C05460=1089.469,232.311,-75.849,176.386,20.960,153.192
C05461=1089.476,232.559,-75.874,176.389,20.962,153.192
C05462=1089.481,232.808,-75.901,176.392,20.965,153.192
C05463=1089.486,233.056,-75.926,176.394,20.967,153.192
C05464=1089.492,233.305,-75.952,176.398,20.970,153.192
C05465=1089.498,233.554,-75.977,176.400,20.972,153.192
C05466=1089.504,233.802,-76.004,176.403,20.974,153.192
C05467=1089.509,234.051,-76.030,176.406,20.977,153.192
C05468=1089.514,234.299,-76.056,176.409,20.979,153.192
C05469=1089.520,234.547,-76.082,176.412,20.981,153.192
C05470=1089.525,234.796,-76.108,176.414,20.984,153.192
C05471=1089.531,235.045,-76.134,176.417,20.986,153.192
C05472=1089.537,235.294,-76.160,176.420,20.989,153.192
C05473=1089.545,235.671,-76.200,176.424,20.992,153.193
C05474=1089.554,236.049,-76.239,176.429,20.996,153.193
C05475=1089.562,236.426,-76.279,176.433,20.999,153.193
C05476=1089.571,236.805,-76.319,176.437,21.003,153.193
C05477=1089.577,237.053,-76.345,176.440,21.006,153.193
C05478=1089.583,237.302,-76.371,176.443,21.008,153.193
C05479=1089.588,237.551,-76.397,176.445,21.010,153.193
C05480=1089.593,237.798,-76.424,176.448,21.013,153.193
C05481=1089.599,238.047,-76.449,176.452,21.015,153.193
C05482=1089.605,238.296,-76.476,176.454,21.017,153.193
C05483=1089.610,238.545,-76.502,176.457,21.020,153.193
C05484=1089.616,238.793,-76.529,176.459,21.022,153.193
C05485=1089.621,239.042,-76.555,176.463,21.025,153.193
C05486=1089.627,239.290,-76.581,176.466,21.027,153.193
C05487=1089.633,239.539,-76.607,176.468,21.029,153.194
C05488=1089.638,239.788,-76.634,176.471,21.032,153.194
C05489=1089.644,240.036,-76.661,176.475,21.034,153.194
C05490=1089.650,240.285,-76.686,176.477,21.036,153.194
C05491=1089.655,240.533,-76.713,176.480,21.039,153.194
C05492=1089.661,240.782,-76.739,176.483,21.042,153.194
C05493=1089.667,241.031,-76.766,176.486,21.043,153.194
C05494=1089.672,241.279,-76.792,176.489,21.046,153.194
C05495=1089.678,241.527,-76.819,176.491,21.048,153.194
C05496=1089.684,241.776,-76.845,176.494,21.051,153.194
C05497=1089.689,242.025,-76.872,176.497,21.054,153.194
C05498=1089.695,242.273,-76.898,176.500,21.056,153.194
C05499=1089.701,242.522,-76.924,176.503,21.058,153.194
C05500=1089.706,242.770,-76.951,176.506,21.060,153.194
C05501=1089.712,243.019,-76.977,176.508,21.063,153.195
C05502=1089.718,243.267,-77.004,176.511,21.065,153.195
C05503=1089.724,243.516,-77.031,176.515,21.068,153.195
C05504=1089.729,243.765,-77.057,176.517,21.070,153.195
C05505=1089.734,244.013,-77.084,176.520,21.073,153.195
C05506=1089.740,244.262,-77.111,176.523,21.075,153.195
C05507=1089.746,244.510,-77.137,176.526,21.077,153.195
C05508=1089.752,244.758,-77.164,176.529,21.080,153.195
C05509=1089.757,245.007,-77.191,176.532,21.083,153.195
C05510=1089.762,245.256,-77.217,176.534,21.085,153.195
C05511=1089.768,245.504,-77.244,176.537,21.088,153.195
C05512=1089.774,245.753,-77.270,176.540,21.090,153.195
C05513=1089.779,246.001,-77.297,176.543,21.092,153.195
C05514=1089.784,246.250,-77.324,176.546,21.095,153.196
C05515=1089.790,246.498,-77.351,176.549,21.097,153.196
C05516=1089.796,246.746,-77.377,176.551,21.099,153.196
C05517=1089.802,246.996,-77.405,176.554,21.102,153.196
C05518=1089.807,247.244,-77.432,176.558,21.104,153.196
C05519=1089.813,247.492,-77.458,176.560,21.107,153.196
C05520=1089.818,247.741,-77.486,176.563,21.109,153.196
C05521=1089.824,247.989,-77.512,176.566,21.112,153.196
C05522=1089.830,248.238,-77.539,176.569,21.115,153.196
C05523=1089.835,248.487,-77.566,176.572,21.117,153.196
C05524=1089.841,248.735,-77.593,176.575,21.119,153.196
C05525=1089.849,249.106,-77.634,176.579,21.123,153.196
C05526=1089.857,249.476,-77.674,176.583,21.127,153.197
C05527=1089.865,249.847,-77.714,176.588,21.131,153.197
C05528=1089.874,250.218,-77.754,176.592,21.134,153.197
C05529=1089.879,250.467,-77.782,176.595,21.137,153.197
C05530=1089.885,250.715,-77.808,176.597,21.139,153.197
C05531=1089.890,250.963,-77.836,176.601,21.142,153.197
C05532=1089.896,251.212,-77.863,176.604,21.145,153.197
C05533=1089.901,251.460,-77.890,176.607,21.147,153.197
C05534=1089.907,251.710,-77.917,176.609,21.149,153.197
C05535=1089.912,251.958,-77.944,176.612,21.152,153.197
C05536=1089.918,252.206,-77.972,176.615,21.155,153.198
C05537=1089.923,252.455,-77.999,176.618,21.157,153.198
C05538=1089.929,252.703,-78.026,176.621,21.160,153.198
C05539=1089.934,252.951,-78.054,176.624,21.162,153.198
C05540=1089.941,253.200,-78.081,176.627,21.164,153.198
C05541=1089.946,253.449,-78.108,176.629,21.167,153.198
C05542=1089.952,253.696,-78.135,176.633,21.169,153.198
C05543=1089.957,253.945,-78.163,176.636,21.172,153.198
C05544=1089.963,254.194,-78.190,176.639,21.175,153.198
C05545=1089.969,254.442,-78.218,176.641,21.177,153.198
C05546=1089.974,254.691,-78.244,176.644,21.179,153.198
C05547=1089.980,254.939,-78.272,176.647,21.182,153.199
C05548=1089.986,255.187,-78.299,176.650,21.184,153.199
C05549=1089.991,255.436,-78.326,176.653,21.187,153.199
C05550=1089.996,255.684,-78.354,176.656,21.190,153.199
C05551=1090.002,255.933,-78.381,176.659,21.192,153.199
C05552=1090.008,256.182,-78.409,176.661,21.194,153.199
C05553=1090.014,256.430,-78.436,176.665,21.197,153.199
C05554=1090.019,256.678,-78.464,176.668,21.200,153.199
C05555=1090.024,256.927,-78.491,176.671,21.202,153.199
C05556=1090.031,257.175,-78.519,176.673,21.205,153.199
C05557=1090.036,257.424,-78.546,176.676,21.207,153.199
C05558=1090.042,257.671,-78.573,176.679,21.210,153.200
C05559=1090.048,257.921,-78.601,176.683,21.212,153.200
C05560=1090.053,258.169,-78.629,176.685,21.215,153.200
C05561=1090.059,258.417,-78.656,176.688,21.217,153.200
C05562=1090.065,258.666,-78.684,176.691,21.219,153.200
C05563=1090.070,258.914,-78.712,176.694,21.222,153.200
C05564=1090.076,259.162,-78.739,176.697,21.224,153.200
C05565=1090.082,259.411,-78.767,176.700,21.227,153.200
C05566=1090.088,259.659,-78.794,176.703,21.230,153.200
C05567=1090.094,259.908,-78.823,176.706,21.232,153.200
C05568=1090.099,260.156,-78.850,176.709,21.235,153.200
C05569=1090.105,260.404,-78.877,176.711,21.237,153.201
C05570=1090.111,260.653,-78.906,176.715,21.240,153.201
C05571=1090.116,260.902,-78.933,176.718,21.242,153.201
C05572=1090.123,261.150,-78.961,176.721,21.245,153.201
C05573=1090.128,261.398,-78.989,176.723,21.247,153.201
C05574=1090.133,261.646,-79.016,176.726,21.250,153.201
C05575=1090.139,261.895,-79.045,176.730,21.252,153.201
C05576=1090.145,262.143,-79.071,176.733,21.255,153.201
C05577=1090.153,262.511,-79.114,176.736,21.259,153.201
C05578=1090.163,262.879,-79.155,176.741,21.262,153.201
C05579=1090.171,263.247,-79.195,176.746,21.266,153.202
C05580=1090.179,263.615,-79.237,176.750,21.270,153.202
C05581=1090.185,263.863,-79.265,176.753,21.273,153.202
C05582=1090.191,264.112,-79.293,176.756,21.275,153.202
C05583=1090.197,264.360,-79.320,176.759,21.277,153.202
C05584=1090.203,264.609,-79.349,176.762,21.280,153.202
C05585=1090.208,264.857,-79.377,176.765,21.283,153.202
C05586=1090.214,265.106,-79.405,176.768,21.285,153.202
C05587=1090.219,265.354,-79.433,176.771,21.288,153.202
C05588=1090.225,265.602,-79.461,176.773,21.290,153.203
C05589=1090.230,265.850,-79.489,176.776,21.293,153.203
C05590=1090.236,266.098,-79.517,176.779,21.296,153.203
C05591=1090.242,266.347,-79.546,176.783,21.298,153.203
C05592=1090.247,266.595,-79.574,176.786,21.301,153.203
C05593=1090.253,266.844,-79.602,176.789,21.304,153.203
C05594=1090.258,267.092,-79.630,176.791,21.306,153.203
C05595=1090.264,267.341,-79.658,176.794,21.309,153.203
C05596=1090.270,267.589,-79.686,176.797,21.311,153.203
C05597=1090.276,267.837,-79.715,176.800,21.314,153.204
C05598=1090.281,268.085,-79.743,176.803,21.317,153.204
C05599=1090.287,268.334,-79.771,176.806,21.319,153.204
C05600=1090.293,268.582,-79.799,176.809,21.322,153.204
C05601=1090.299,268.831,-79.828,176.812,21.325,153.204
C05602=1090.304,269.079,-79.856,176.815,21.327,153.204
C05603=1090.310,269.327,-79.885,176.818,21.330,153.204
C05604=1090.316,269.576,-79.913,176.822,21.332,153.204
C05605=1090.321,269.824,-79.941,176.824,21.335,153.204
C05606=1090.327,270.073,-79.970,176.827,21.337,153.205
C05607=1090.332,270.320,-79.999,176.830,21.340,153.205
C05608=1090.338,270.569,-80.027,176.833,21.343,153.205
C05609=1090.344,270.817,-80.055,176.836,21.346,153.205
C05610=1090.349,271.066,-80.083,176.839,21.348,153.205
C05611=1090.355,271.313,-80.112,176.841,21.350,153.205
C05612=1090.360,271.562,-80.141,176.845,21.353,153.205
C05613=1090.366,271.811,-80.169,176.848,21.356,153.205
C05614=1090.372,272.058,-80.198,176.851,21.359,153.206
C05615=1090.378,272.307,-80.226,176.854,21.362,153.206
C05616=1090.383,272.554,-80.255,176.857,21.364,153.206
C05617=1090.389,272.803,-80.283,176.860,21.367,153.206
C05618=1090.395,273.052,-80.312,176.862,21.369,153.206
C05619=1090.400,273.300,-80.341,176.865,21.372,153.206
C05620=1090.406,273.548,-80.369,176.869,21.375,153.206
C05621=1090.412,273.796,-80.398,176.872,21.377,153.206
C05622=1090.417,274.045,-80.427,176.875,21.380,153.207
C05623=1090.423,274.293,-80.456,176.878,21.383,153.207
C05624=1090.429,274.541,-80.484,176.881,21.386,153.207
C05625=1090.434,274.790,-80.513,176.883,21.388,153.207
C05626=1090.440,275.038,-80.542,176.886,21.391,153.207
C05627=1090.446,275.286,-80.570,176.889,21.394,153.207
C05628=1090.451,275.535,-80.599,176.893,21.396,153.207
C05629=1090.460,275.905,-80.642,176.897,21.400,153.208
C05630=1090.468,276.275,-80.685,176.902,21.405,153.208
C05631=1090.477,276.646,-80.729,176.906,21.408,153.208
C05632=1090.485,277.018,-80.771,176.910,21.412,153.208
C05633=1090.491,277.266,-80.801,176.913,21.415,153.208
C05634=1090.496,277.514,-80.829,176.916,21.418,153.209
C05635=1090.502,277.763,-80.858,176.920,21.421,153.209
C05636=1090.508,278.011,-80.887,176.923,21.423,153.209
C05637=1090.514,278.258,-80.916,176.926,21.426,153.209
C05638=1090.519,278.507,-80.946,176.928,21.429,153.209
C05639=1090.525,278.755,-80.974,176.931,21.432,153.209
C05640=1090.530,279.003,-81.003,176.934,21.435,153.209
C05641=1090.536,279.251,-81.032,176.937,21.437,153.209
C05642=1090.542,279.500,-81.062,176.940,21.440,153.210
C05643=1090.548,279.748,-81.090,176.943,21.443,153.210
C05644=1090.553,279.996,-81.119,176.946,21.446,153.210
C05645=1090.559,280.244,-81.149,176.949,21.448,153.210
C05646=1090.564,280.493,-81.178,176.953,21.451,153.210
C05647=1090.571,280.741,-81.207,176.956,21.454,153.210
C05648=1090.576,280.989,-81.237,176.958,21.456,153.211
C05649=1090.581,281.237,-81.265,176.961,21.459,153.211
C05650=1090.587,281.486,-81.294,176.964,21.462,153.211
C05651=1090.593,281.734,-81.323,176.967,21.465,153.211
C05652=1090.599,281.982,-81.353,176.970,21.468,153.211
C05653=1090.604,282.230,-81.382,176.973,21.470,153.211
C05654=1090.610,282.478,-81.411,176.976,21.473,153.212
C05655=1090.615,282.727,-81.441,176.979,21.476,153.212
C05656=1090.621,282.975,-81.471,176.982,21.479,153.212
C05657=1090.627,283.223,-81.499,176.985,21.482,153.212
C05658=1090.632,283.471,-81.529,176.988,21.485,153.212
C05659=1090.638,283.719,-81.559,176.991,21.488,153.212
C05660=1090.644,283.968,-81.588,176.994,21.491,153.213
C05661=1090.649,284.216,-81.617,176.997,21.493,153.213
C05662=1090.654,284.464,-81.647,177.000,21.495,153.213
C05663=1090.660,284.712,-81.676,177.003,21.498,153.213
C05664=1090.666,284.960,-81.705,177.006,21.501,153.213
C05665=1090.672,285.209,-81.735,177.009,21.504,153.213
C05666=1090.678,285.456,-81.765,177.012,21.507,153.213
C05667=1090.684,285.705,-81.794,177.015,21.510,153.214
C05668=1090.688,285.952,-81.824,177.018,21.513,153.214
C05669=1090.694,286.201,-81.853,177.021,21.515,153.214
C05670=1090.700,286.449,-81.882,177.024,21.518,153.214
C05671=1090.706,286.697,-81.912,177.027,21.521,153.214
C05672=1090.712,286.945,-81.942,177.030,21.524,153.214
C05673=1090.717,287.194,-81.972,177.034,21.527,153.215
C05674=1090.723,287.442,-82.001,177.037,21.530,153.215
C05675=1090.729,287.690,-82.030,177.040,21.533,153.215
C05676=1090.735,287.938,-82.061,177.043,21.536,153.215
C05677=1090.740,288.187,-82.090,177.046,21.538,153.215
C05678=1090.746,288.434,-82.119,177.049,21.541,153.215
C05679=1090.752,288.682,-82.150,177.052,21.544,153.216
C05680=1090.757,288.930,-82.179,177.055,21.547,153.216
C05681=1090.766,289.311,-82.225,177.060,21.551,153.216
C05682=1090.775,289.691,-82.270,177.064,21.556,153.216
C05683=1090.784,290.071,-82.316,177.068,21.560,153.217
C05684=1090.792,290.452,-82.362,177.073,21.565,153.217
C05685=1090.798,290.700,-82.392,177.076,21.568,153.217
C05686=1090.804,290.948,-82.422,177.079,21.570,153.217
C05687=1090.809,291.196,-82.452,177.082,21.573,153.217
C05688=1090.815,291.444,-82.482,177.085,21.576,153.218
C05689=1090.821,291.693,-82.512,177.088,21.580,153.218
C05690=1090.826,291.940,-82.542,177.091,21.582,153.218
C05691=1090.832,292.189,-82.572,177.094,21.585,153.218
C05692=1090.838,292.437,-82.602,177.097,21.588,153.218
C05693=1090.843,292.685,-82.632,177.100,21.591,153.219
C05694=1090.849,292.933,-82.662,177.103,21.594,153.219
C05695=1090.855,293.181,-82.691,177.107,21.597,153.219
C05696=1090.860,293.429,-82.722,177.109,21.600,153.219
C05697=1090.866,293.677,-82.752,177.112,21.603,153.219
C05698=1090.872,293.925,-82.782,177.116,21.606,153.220
C05699=1090.878,294.173,-82.812,177.119,21.609,153.220
C05700=1090.883,294.421,-82.843,177.122,21.612,153.220
C05701=1090.889,294.670,-82.872,177.124,21.615,153.220
C05702=1090.895,294.917,-82.903,177.128,21.618,153.220
C05703=1090.901,295.165,-82.933,177.131,21.621,153.221
C05704=1090.906,295.414,-82.963,177.134,21.623,153.221
C05705=1090.912,295.661,-82.993,177.137,21.626,153.221
C05706=1090.918,295.909,-83.023,177.140,21.630,153.221
C05707=1090.923,296.157,-83.054,177.143,21.633,153.221
C05708=1090.929,296.406,-83.083,177.146,21.635,153.222
C05709=1090.935,296.653,-83.114,177.149,21.638,153.222
C05710=1090.940,296.902,-83.144,177.152,21.642,153.222
C05711=1090.946,297.149,-83.175,177.155,21.644,153.222
C05712=1090.952,297.397,-83.205,177.158,21.647,153.222
C05713=1090.958,297.646,-83.235,177.161,21.651,153.223
C05714=1090.963,297.894,-83.266,177.164,21.653,153.223
C05715=1090.969,298.142,-83.296,177.167,21.656,153.223
C05716=1090.974,298.390,-83.327,177.170,21.660,153.223
C05717=1090.980,298.638,-83.357,177.173,21.663,153.224
C05718=1090.985,298.886,-83.388,177.176,21.666,153.224
C05719=1090.991,299.134,-83.418,177.179,21.669,153.224
C05720=1090.997,299.382,-83.449,177.182,21.673,153.224
C05721=1091.002,299.630,-83.480,177.185,21.675,153.225
C05722=1091.008,299.878,-83.510,177.188,21.679,153.225
C05723=1091.013,300.126,-83.541,177.191,21.682,153.225
C05724=1091.019,300.374,-83.571,177.194,21.685,153.225
C05725=1091.025,300.622,-83.602,177.197,21.688,153.226
C05726=1091.030,300.870,-83.633,177.200,21.691,153.226
C05727=1091.036,301.118,-83.663,177.203,21.694,153.226
C05728=1091.041,301.366,-83.694,177.206,21.697,153.226
C05729=1091.047,301.614,-83.725,177.209,21.700,153.227
C05730=1091.053,301.862,-83.755,177.212,21.703,153.227
C05731=1091.058,302.110,-83.786,177.215,21.706,153.227
C05732=1091.064,302.358,-83.816,177.218,21.710,153.227
C05733=1091.072,302.726,-83.862,177.223,21.714,153.228
C05734=1091.080,303.094,-83.909,177.228,21.719,153.228
C05735=1091.088,303.462,-83.954,177.232,21.724,153.228
C05736=1091.097,303.830,-84.000,177.237,21.729,153.229
C05737=1091.102,304.078,-84.031,177.240,21.732,153.229
C05738=1091.109,304.326,-84.061,177.243,21.735,153.229
C05739=1091.114,304.574,-84.092,177.246,21.738,153.229
C05740=1091.120,304.822,-84.123,177.249,21.741,153.230
C05741=1091.125,305.070,-84.154,177.251,21.744,153.230
C05742=1091.131,305.318,-84.185,177.254,21.747,153.230
C05743=1091.137,305.566,-84.217,177.257,21.751,153.231
C05744=1091.143,305.814,-84.247,177.261,21.754,153.231
C05745=1091.149,306.088,-84.281,177.264,21.757,153.231
C05746=1091.155,306.362,-84.316,177.268,21.761,153.231
C05747=1091.162,306.637,-84.350,177.271,21.764,153.232
C05748=1091.168,306.910,-84.384,177.274,21.768,153.232
C05749=1091.173,307.158,-84.415,177.278,21.771,153.232
C05750=1091.179,307.407,-84.447,177.280,21.774,153.232
C05751=1091.185,307.654,-84.478,177.283,21.778,153.233
C05752=1091.190,307.902,-84.509,177.286,21.780,153.233
C05753=1091.197,308.150,-84.540,177.289,21.784,153.233
C05754=1091.202,308.398,-84.571,177.293,21.788,153.234
C05755=1091.208,308.646,-84.602,177.296,21.790,153.234
C05756=1091.214,308.894,-84.633,177.299,21.794,153.234
C05757=1091.219,309.142,-84.665,177.302,21.797,153.234
C05758=1091.225,309.391,-84.696,177.305,21.800,153.234
C05759=1091.231,309.638,-84.727,177.308,21.803,153.235
C05760=1091.237,309.885,-84.759,177.311,21.807,153.235
C05761=1091.243,310.134,-84.790,177.315,21.810,153.235
C05762=1091.248,310.382,-84.822,177.317,21.813,153.236
C05763=1091.254,310.630,-84.852,177.320,21.816,153.236
C05764=1091.260,310.878,-84.884,177.323,21.819,153.236
C05765=1091.265,311.125,-84.916,177.326,21.823,153.236
C05766=1091.272,311.374,-84.946,177.329,21.826,153.237
C05767=1091.277,311.621,-84.978,177.332,21.829,153.237
C05768=1091.283,311.869,-85.010,177.336,21.833,153.237
C05769=1091.289,312.117,-85.040,177.339,21.836,153.238
C05770=1091.295,312.365,-85.072,177.342,21.839,153.238
C05771=1091.300,312.613,-85.104,177.345,21.842,153.238
C05772=1091.307,312.861,-85.135,177.348,21.845,153.238
C05773=1091.312,313.109,-85.166,177.351,21.849,153.239
C05774=1091.318,313.357,-85.198,177.355,21.852,153.239
C05775=1091.323,313.605,-85.230,177.357,21.855,153.239
C05776=1091.330,313.853,-85.261,177.360,21.859,153.239
C05777=1091.335,314.101,-85.292,177.363,21.862,153.240
C05778=1091.341,314.349,-85.324,177.366,21.865,153.240
C05779=1091.347,314.596,-85.356,177.369,21.868,153.240
C05780=1091.353,314.844,-85.388,177.373,21.872,153.241
C05781=1091.359,315.093,-85.420,177.376,21.875,153.241
C05782=1091.365,315.340,-85.451,177.379,21.879,153.241
C05783=1091.370,315.588,-85.483,177.382,21.882,153.242
C05784=1091.376,315.836,-85.515,177.384,21.885,153.242
C05785=1091.385,316.232,-85.566,177.390,21.891,153.242
C05786=1091.394,316.630,-85.617,177.395,21.896,153.243
C05787=1091.403,317.027,-85.668,177.399,21.902,153.243
C05788=1091.412,317.424,-85.718,177.404,21.907,153.244
C05789=1091.418,317.672,-85.750,177.407,21.911,153.244
C05790=1091.422,317.920,-85.782,177.411,21.914,153.245
C05791=1091.428,318.168,-85.815,177.413,21.918,153.245
C05792=1091.434,318.415,-85.847,177.416,21.922,153.245
C05793=1091.440,318.663,-85.879,177.419,21.925,153.246
C05794=1091.445,318.910,-85.911,177.422,21.928,153.246
C05795=1091.451,319.159,-85.943,177.426,21.932,153.246
C05796=1091.457,319.407,-85.975,177.428,21.936,153.247
C05797=1091.462,319.655,-86.007,177.431,21.939,153.247
C05798=1091.468,319.903,-86.039,177.434,21.942,153.247
C05799=1091.473,320.150,-86.071,177.437,21.946,153.248
C05800=1091.480,320.398,-86.103,177.441,21.950,153.248
C05801=1091.486,320.646,-86.135,177.443,21.953,153.248
C05802=1091.491,320.894,-86.167,177.446,21.956,153.249
C05803=1091.496,321.142,-86.200,177.449,21.960,153.249
C05804=1091.502,321.389,-86.232,177.453,21.964,153.250
C05805=1091.508,321.637,-86.264,177.456,21.967,153.250
C05806=1091.514,321.886,-86.296,177.459,21.971,153.250
C05807=1091.519,322.133,-86.328,177.461,21.974,153.250
C05808=1091.525,322.381,-86.361,177.465,21.978,153.251
C05809=1091.531,322.629,-86.393,177.468,21.981,153.251
C05810=1091.536,322.877,-86.425,177.471,21.985,153.252
C05811=1091.542,323.124,-86.457,177.474,21.988,153.252
C05812=1091.548,323.373,-86.490,177.477,21.992,153.252
C05813=1091.553,323.620,-86.522,177.480,21.996,153.253
C05814=1091.559,323.868,-86.555,177.483,21.999,153.253
C05815=1091.565,324.116,-86.587,177.486,22.003,153.253
C05816=1091.571,324.364,-86.620,177.490,22.006,153.254
C05817=1091.576,324.612,-86.652,177.492,22.010,153.254
C05818=1091.583,324.859,-86.684,177.495,22.013,153.254
C05819=1091.588,325.108,-86.717,177.498,22.017,153.255
C05820=1091.594,325.355,-86.750,177.502,22.021,153.255
C05821=1091.600,325.603,-86.781,177.504,22.024,153.256
C05822=1091.606,325.850,-86.814,177.507,22.028,153.256
C05823=1091.611,326.099,-86.847,177.511,22.032,153.256
C05824=1091.617,326.347,-86.879,177.514,22.035,153.257
C05825=1091.623,326.595,-86.911,177.517,22.039,153.257
C05826=1091.628,326.842,-86.944,177.519,22.042,153.257
C05827=1091.635,327.090,-86.977,177.523,22.046,153.258
C05828=1091.641,327.338,-87.009,177.526,22.050,153.258
C05829=1091.646,327.586,-87.043,177.529,22.053,153.259
C05830=1091.652,327.834,-87.075,177.532,22.057,153.259
C05831=1091.657,328.081,-87.108,177.535,22.061,153.259
C05832=1091.663,328.329,-87.140,177.538,22.064,153.260
C05833=1091.669,328.577,-87.172,177.542,22.068,153.260
C05834=1091.675,328.825,-87.206,177.544,22.072,153.260
C05835=1091.681,329.072,-87.238,177.547,22.076,153.261
C05836=1091.687,329.320,-87.271,177.551,22.079,153.261
C05837=1091.697,329.710,-87.323,177.555,22.085,153.262
C05838=1091.706,330.100,-87.374,177.560,22.091,153.262
C05839=1091.714,330.490,-87.426,177.565,22.097,153.263
C05840=1091.724,330.880,-87.478,177.570,22.102,153.264
C05841=1091.730,331.128,-87.511,177.573,22.106,153.264
C05842=1091.736,331.375,-87.543,177.576,22.110,153.265
C05843=1091.742,331.623,-87.577,177.579,22.114,153.265
C05844=1091.748,331.871,-87.610,177.582,22.117,153.265
C05845=1091.753,332.120,-87.642,177.585,22.121,153.266
C05846=1091.759,332.367,-87.675,177.589,22.125,153.266
C05847=1091.765,332.615,-87.708,177.591,22.129,153.267
C05848=1091.771,332.863,-87.742,177.595,22.133,153.267
C05849=1091.776,333.110,-87.775,177.598,22.137,153.267
C05850=1091.782,333.358,-87.807,177.600,22.140,153.268
C05851=1091.787,333.606,-87.841,177.604,22.145,153.268
C05852=1091.793,333.854,-87.874,177.607,22.148,153.269
C05853=1091.799,334.101,-87.907,177.609,22.152,153.269
C05854=1091.805,334.349,-87.940,177.613,22.156,153.270
C05855=1091.811,334.596,-87.974,177.616,22.160,153.270
C05856=1091.816,334.844,-88.007,177.619,22.164,153.271
C05857=1091.823,335.092,-88.040,177.622,22.168,153.271
C05858=1091.828,335.340,-88.073,177.625,22.171,153.271
C05859=1091.834,335.588,-88.107,177.628,22.175,153.272
C05860=1091.839,335.836,-88.140,177.631,22.179,153.272
C05861=1091.846,336.083,-88.173,177.635,22.183,153.273
C05862=1091.851,336.330,-88.207,177.637,22.187,153.273
C05863=1091.857,336.578,-88.240,177.640,22.191,153.274
C05864=1091.862,336.826,-88.274,177.644,22.195,153.274
C05865=1091.868,337.074,-88.307,177.646,22.199,153.275
C05866=1091.874,337.322,-88.340,177.650,22.203,153.275
C05867=1091.880,337.569,-88.374,177.653,22.207,153.276
C05868=1091.886,337.817,-88.407,177.655,22.211,153.276
C05869=1091.891,338.065,-88.440,177.659,22.215,153.277
C05870=1091.897,338.312,-88.474,177.662,22.219,153.277
C05871=1091.903,338.560,-88.507,177.665,22.223,153.277
C05872=1091.909,338.808,-88.541,177.668,22.227,153.278
C05873=1091.915,339.056,-88.575,177.671,22.231,153.278
C05874=1091.921,339.303,-88.608,177.674,22.235,153.279
C05875=1091.927,339.551,-88.642,177.677,22.239,153.279
C05876=1091.932,339.799,-88.676,177.680,22.243,153.280
C05877=1091.938,340.047,-88.709,177.683,22.247,153.280
C05878=1091.944,340.294,-88.743,177.686,22.252,153.281
C05879=1091.949,340.542,-88.776,177.689,22.255,153.281
C05880=1091.955,340.789,-88.810,177.693,22.260,153.282
C05881=1091.961,341.037,-88.844,177.695,22.264,153.282
C05882=1091.967,341.284,-88.878,177.699,22.268,153.283
C05883=1091.972,341.532,-88.911,177.702,22.272,153.283
C05884=1091.978,341.779,-88.945,177.705,22.276,153.284
C05885=1091.984,342.028,-88.979,177.708,22.280,153.284
C05886=1091.990,342.275,-89.013,177.710,22.284,153.285
C05887=1091.996,342.523,-89.047,177.714,22.289,153.285
C05888=1092.002,342.770,-89.080,177.717,22.292,153.286
C05889=1092.011,343.154,-89.133,177.721,22.299,153.287
C05890=1092.019,343.539,-89.186,177.726,22.305,153.288
C05891=1092.028,343.923,-89.238,177.731,22.312,153.288
C05892=1092.037,344.307,-89.291,177.736,22.318,153.289
C05893=1092.044,344.555,-89.326,177.739,22.323,153.290
C05894=1092.049,344.802,-89.359,177.742,22.327,153.290
C05895=1092.055,345.050,-89.393,177.745,22.331,153.291
C05896=1092.061,345.297,-89.427,177.748,22.336,153.291
C05897=1092.066,345.545,-89.462,177.751,22.340,153.292
C05898=1092.072,345.793,-89.495,177.754,22.344,153.292
C05899=1092.078,346.040,-89.530,177.757,22.349,153.293
C05900=1092.084,346.288,-89.564,177.760,22.352,153.293
C05901=1092.089,346.535,-89.598,177.764,22.357,153.294
C05902=1092.096,346.783,-89.633,177.766,22.361,153.295
C05903=1092.101,347.031,-89.667,177.770,22.366,153.295
C05904=1092.107,347.278,-89.701,177.772,22.370,153.296
C05905=1092.112,347.525,-89.735,177.776,22.374,153.296
C05906=1092.118,347.773,-89.769,177.779,22.379,153.297
C05907=1092.125,348.021,-89.804,177.782,22.383,153.297
C05908=1092.130,348.268,-89.839,177.785,22.388,153.298
C05909=1092.136,348.516,-89.873,177.788,22.392,153.299
C05910=1092.142,348.764,-89.907,177.791,22.396,153.299
C05911=1092.147,349.011,-89.942,177.794,22.400,153.300
C05912=1092.153,349.258,-89.976,177.797,22.405,153.300
C05913=1092.159,349.506,-90.010,177.800,22.409,153.301
C05914=1092.165,349.754,-90.045,177.803,22.414,153.301
C05915=1092.171,350.001,-90.079,177.807,22.418,153.302
C05916=1092.177,350.249,-90.113,177.809,22.423,153.303
C05917=1092.182,350.497,-90.148,177.813,22.427,153.303
C05918=1092.188,350.744,-90.182,177.815,22.431,153.304
C05919=1092.194,350.991,-90.217,177.819,22.436,153.304
C05920=1092.200,351.239,-90.252,177.821,22.440,153.305
C05921=1092.206,351.486,-90.286,177.825,22.445,153.306
C05922=1092.211,351.734,-90.320,177.828,22.450,153.306
C05923=1092.217,351.982,-90.355,177.831,22.454,153.307
C05924=1092.223,352.229,-90.390,177.834,22.459,153.307
C05925=1092.229,352.477,-90.425,177.836,22.463,153.308
C05926=1092.234,352.725,-90.459,177.840,22.468,153.309
C05927=1092.240,352.972,-90.493,177.843,22.472,153.309
C05928=1092.246,353.220,-90.529,177.846,22.476,153.310
C05929=1092.252,353.467,-90.563,177.849,22.482,153.311
C05930=1092.258,353.715,-90.599,177.852,22.486,153.311
C05931=1092.264,353.962,-90.633,177.855,22.490,153.312
C05932=1092.269,354.209,-90.668,177.859,22.495,153.312
C05933=1092.276,354.457,-90.703,177.861,22.500,153.313
C05934=1092.281,354.704,-90.737,177.864,22.504,153.314
C05935=1092.287,354.952,-90.773,177.868,22.509,153.314
C05936=1092.293,355.199,-90.807,177.870,22.514,153.315
C05937=1092.298,355.446,-90.842,177.874,22.518,153.316
C05938=1092.305,355.694,-90.877,177.877,22.523,153.316
C05939=1092.310,355.941,-90.912,177.879,22.527,153.317
C05940=1092.316,356.190,-90.947,177.883,22.532,153.318
C05941=1092.325,356.576,-91.002,177.887,22.540,153.319
C05942=1092.334,356.962,-91.057,177.892,22.547,153.320
C05943=1092.343,357.349,-91.112,177.897,22.555,153.321
C05944=1092.353,357.736,-91.166,177.902,22.562,153.322
C05945=1092.358,357.983,-91.201,177.905,22.567,153.322
C05946=1092.364,358.231,-91.237,177.907,22.571,153.323
C05947=1092.370,358.478,-91.272,177.911,22.576,153.324
C05948=1092.376,358.726,-91.306,177.914,22.581,153.324
C05949=1092.382,358.973,-91.342,177.916,22.586,153.325
C05950=1092.388,359.220,-91.378,177.920,22.591,153.326
C05951=1092.394,359.468,-91.412,177.923,22.595,153.327
C05952=1092.400,359.715,-91.447,177.926,22.600,153.327
C05953=1092.405,359.962,-91.483,177.929,22.605,153.328
C05954=1092.411,360.210,-91.518,177.932,22.610,153.329
C05955=1092.417,360.458,-91.554,177.936,22.615,153.329
C05956=1092.423,360.704,-91.589,177.938,22.619,153.330
C05957=1092.429,360.953,-91.624,177.941,22.624,153.331
C05958=1092.434,361.200,-91.659,177.945,22.630,153.331
C05959=1092.440,361.447,-91.695,177.947,22.634,153.332
C05960=1092.446,361.694,-91.730,177.950,22.639,153.333
C05961=1092.452,361.942,-91.766,177.953,22.644,153.334
C05962=1092.457,362.189,-91.802,177.957,22.649,153.334
C05963=1092.463,362.437,-91.837,177.959,22.654,153.335
C05964=1092.470,362.684,-91.872,177.962,22.659,153.336
C05965=1092.476,362.931,-91.908,177.966,22.664,153.337
C05966=1092.482,363.179,-91.943,177.968,22.669,153.337
C05967=1092.488,363.426,-91.979,177.971,22.674,153.338
C05968=1092.493,363.673,-92.015,177.974,22.679,153.339
C05969=1092.499,363.921,-92.050,177.978,22.684,153.340
C05970=1092.504,364.168,-92.086,177.980,22.689,153.340
C05971=1092.511,364.416,-92.121,177.983,22.694,153.341
C05972=1092.517,364.663,-92.158,177.987,22.700,153.342
C05973=1092.522,364.910,-92.193,177.990,22.705,153.343
C05974=1092.528,365.157,-92.229,177.992,22.709,153.343
C05975=1092.534,365.405,-92.265,177.996,22.714,153.344
C05976=1092.540,365.652,-92.300,177.999,22.720,153.345
C05977=1092.546,365.899,-92.336,178.002,22.725,153.346
C05978=1092.552,366.147,-92.372,178.005,22.730,153.347
C05979=1092.558,366.394,-92.408,178.007,22.735,153.347
C05980=1092.563,366.642,-92.444,178.011,22.741,153.348
C05981=1092.569,366.889,-92.480,178.014,22.746,153.349
C05982=1092.575,367.136,-92.516,178.017,22.751,153.350
C05983=1092.581,367.383,-92.551,178.020,22.756,153.350
C05984=1092.587,367.630,-92.588,178.022,22.761,153.351
C05985=1092.592,367.877,-92.623,178.026,22.767,153.352
C05986=1092.598,368.125,-92.660,178.029,22.772,153.353
C05987=1092.604,368.372,-92.696,178.032,22.777,153.354
C05988=1092.610,368.620,-92.732,178.035,22.783,153.355
C05989=1092.616,368.866,-92.768,178.038,22.787,153.355
C05990=1092.622,369.114,-92.804,178.041,22.793,153.356
C05991=1092.627,369.362,-92.841,178.044,22.798,153.357
C05992=1092.633,369.609,-92.876,178.047,22.804,153.358
C05993=1092.643,370.011,-92.935,178.052,22.813,153.359
C05994=1092.652,370.412,-92.994,178.057,22.821,153.361
C05995=1092.662,370.815,-93.052,178.061,22.830,153.362
C05996=1092.672,371.217,-93.111,178.066,22.838,153.363
C05997=1092.677,371.464,-93.148,178.069,22.844,153.364
C05998=1092.684,371.711,-93.185,178.072,22.849,153.365
C05999=1092.690,371.959,-93.220,178.075,22.855,153.366
C06000=1092.696,372.206,-93.257,178.079,22.860,153.367
C06001=1092.701,372.452,-93.293,178.082,22.866,153.368
C06002=1092.707,372.700,-93.329,178.085,22.871,153.369
C06003=1092.713,372.947,-93.366,178.087,22.877,153.370
C06004=1092.719,373.195,-93.403,178.090,22.882,153.370
C06005=1092.725,373.442,-93.439,178.093,22.888,153.371
C06006=1092.731,373.689,-93.475,178.096,22.893,153.372
C06007=1092.737,373.937,-93.512,178.099,22.899,153.373
C06008=1092.743,374.184,-93.548,178.103,22.904,153.374
C06009=1092.748,374.430,-93.585,178.106,22.910,153.375
C06010=1092.754,374.677,-93.621,178.109,22.916,153.376
C06011=1092.760,374.925,-93.658,178.112,22.922,153.377
C06012=1092.766,375.172,-93.695,178.114,22.927,153.378
C06013=1092.772,375.419,-93.732,178.117,22.933,153.379
C06014=1092.778,375.667,-93.768,178.120,22.938,153.379
C06015=1092.784,375.914,-93.805,178.123,22.944,153.380
C06016=1092.789,376.161,-93.841,178.126,22.950,153.381
C06017=1092.795,376.408,-93.878,178.129,22.955,153.382
C06018=1092.801,376.655,-93.914,178.132,22.961,153.383
C06019=1092.807,376.902,-93.951,178.135,22.967,153.384
C06020=1092.813,377.150,-93.988,178.138,22.973,153.385
C06021=1092.819,377.396,-94.025,178.141,22.979,153.386
C06022=1092.825,377.644,-94.063,178.144,22.984,153.387
C06023=1092.831,377.891,-94.099,178.147,22.990,153.388
C06024=1092.837,378.138,-94.136,178.150,22.996,153.389
C06025=1092.842,378.385,-94.173,178.153,23.002,153.390
C06026=1092.849,378.632,-94.209,178.156,23.008,153.391
C06027=1092.854,378.880,-94.247,178.159,23.013,153.392
C06028=1092.861,379.126,-94.284,178.162,23.019,153.393
C06029=1092.866,379.374,-94.321,178.165,23.025,153.394
C06030=1092.872,379.621,-94.358,178.168,23.031,153.395
C06031=1092.878,379.868,-94.394,178.171,23.037,153.396
C06032=1092.884,380.115,-94.432,178.174,23.043,153.397
C06033=1092.890,380.362,-94.469,178.177,23.049,153.398
C06034=1092.896,380.609,-94.505,178.180,23.055,153.399
C06035=1092.902,380.856,-94.543,178.183,23.061,153.400
C06036=1092.908,381.103,-94.580,178.186,23.067,153.401
C06037=1092.914,381.350,-94.617,178.189,23.073,153.402
C06038=1092.920,381.597,-94.654,178.192,23.079,153.403
C06039=1092.926,381.844,-94.691,178.195,23.085,153.404
C06040=1092.931,382.091,-94.729,178.198,23.091,153.405
C06041=1092.938,382.338,-94.766,178.201,23.097,153.406
C06042=1092.943,382.586,-94.803,178.204,23.103,153.407
C06043=1092.950,382.833,-94.841,178.207,23.109,153.408
C06044=1092.956,383.080,-94.878,178.210,23.115,153.409
C06045=1092.961,383.294,-94.911,178.212,23.120,153.410
C06046=1092.966,383.509,-94.943,178.215,23.126,153.411
C06047=1092.971,383.724,-94.976,178.217,23.131,153.412
C06048=1092.976,383.939,-95.008,178.219,23.136,153.413
C06049=1092.981,384.154,-95.041,178.223,23.142,153.414
C06050=1092.986,384.368,-95.073,178.225,23.147,153.415
C06051=1092.991,384.583,-95.105,178.228,23.153,153.416
C06052=1092.996,384.798,-95.138,178.230,23.158,153.417
C06053=1093.002,385.044,-95.176,178.233,23.165,153.418
C06054=1093.008,385.291,-95.214,178.236,23.171,153.419
C06055=1093.014,385.539,-95.251,178.239,23.177,153.420
C06056=1093.020,385.786,-95.289,178.241,23.184,153.421
C06057=1093.026,386.033,-95.326,178.244,23.190,153.422
C06058=1093.032,386.279,-95.364,178.248,23.196,153.423
C06059=1093.037,386.527,-95.401,178.251,23.203,153.424
C06060=1093.043,386.774,-95.439,178.254,23.209,153.425
C06061=1093.049,387.020,-95.477,178.257,23.215,153.427
C06062=1093.056,387.268,-95.515,178.260,23.222,153.428
C06063=1093.062,387.514,-95.553,178.262,23.228,153.429
C06064=1093.068,387.761,-95.590,178.265,23.234,153.430
C06065=1093.073,388.009,-95.627,178.268,23.241,153.431
C06066=1093.079,388.255,-95.665,178.272,23.248,153.432
C06067=1093.086,388.503,-95.703,178.274,23.254,153.433
C06068=1093.091,388.750,-95.741,178.277,23.261,153.435
C06069=1093.097,388.996,-95.779,178.280,23.267,153.436
C06070=1093.103,389.243,-95.817,178.283,23.274,153.437
C06071=1093.110,389.490,-95.855,178.286,23.280,153.438
C06072=1093.116,389.737,-95.892,178.289,23.287,153.439
C06073=1093.122,389.984,-95.930,178.292,23.294,153.440
C06074=1093.128,390.231,-95.968,178.295,23.300,153.442
C06075=1093.134,390.478,-96.006,178.298,23.306,153.443
C06076=1093.139,390.725,-96.045,178.301,23.313,153.444
C06077=1093.146,390.972,-96.083,178.303,23.320,153.445
C06078=1093.152,391.219,-96.121,178.307,23.327,153.446
C06079=1093.158,391.465,-96.159,178.310,23.333,153.448
C06080=1093.164,391.713,-96.197,178.313,23.340,153.449
C06081=1093.170,391.960,-96.235,178.315,23.347,153.450
C06082=1093.176,392.206,-96.273,178.318,23.353,153.451
C06083=1093.182,392.454,-96.312,178.322,23.360,153.452
C06084=1093.188,392.700,-96.350,178.324,23.367,153.454
C06085=1093.194,392.947,-96.387,178.327,23.374,153.455
C06086=1093.200,393.194,-96.427,178.330,23.381,153.456
C06087=1093.206,393.441,-96.465,178.333,23.388,153.457
C06088=1093.212,393.688,-96.503,178.336,23.395,153.459
C06089=1093.218,393.935,-96.542,178.339,23.401,153.460
C06090=1093.224,394.182,-96.579,178.342,23.408,153.461
C06091=1093.230,394.429,-96.618,178.345,23.415,153.463
C06092=1093.236,394.675,-96.657,178.348,23.423,153.464
C06093=1093.242,394.923,-96.695,178.350,23.429,153.465
C06094=1093.247,395.170,-96.733,178.353,23.436,153.466
C06095=1093.254,395.417,-96.772,178.357,23.443,153.468
C06096=1093.260,395.664,-96.810,178.359,23.451,153.469
C06097=1093.266,395.910,-96.849,178.362,23.457,153.470
C06098=1093.272,396.157,-96.887,178.365,23.465,153.472
C06099=1093.278,396.404,-96.926,178.368,23.472,153.473
C06100=1093.284,396.651,-96.964,178.371,23.479,153.474
C06101=1093.289,396.872,-96.999,178.374,23.485,153.476
C06102=1093.295,397.093,-97.034,178.375,23.492,153.477
C06103=1093.300,397.315,-97.068,178.378,23.498,153.478
C06104=1093.305,397.535,-97.103,178.381,23.505,153.479
C06105=1093.311,397.757,-97.138,178.384,23.511,153.480
C06106=1093.316,397.978,-97.172,178.386,23.517,153.482
C06107=1093.322,398.200,-97.208,178.389,23.524,153.483
C06108=1093.327,398.421,-97.243,178.391,23.531,153.484
C06109=1093.333,398.668,-97.281,178.394,23.538,153.485
C06110=1093.339,398.915,-97.320,178.398,23.545,153.487
C06111=1093.345,399.161,-97.359,178.400,23.552,153.488
C06112=1093.351,399.409,-97.398,178.403,23.560,153.490
C06113=1093.357,399.655,-97.436,178.406,23.567,153.491
C06114=1093.363,399.902,-97.475,178.409,23.574,153.492
C06115=1093.369,400.149,-97.514,178.412,23.583,153.494
C06116=1093.375,400.396,-97.554,178.415,23.590,153.495
C06117=1093.382,400.643,-97.593,178.417,23.597,153.497
C06118=1093.387,400.889,-97.632,178.421,23.605,153.498
C06119=1093.393,401.137,-97.670,178.423,23.612,153.500
C06120=1093.399,401.383,-97.709,178.426,23.619,153.501
C06121=1093.405,401.630,-97.748,178.429,23.627,153.502
C06122=1093.411,401.877,-97.788,178.432,23.635,153.504
C06123=1093.417,402.124,-97.827,178.435,23.643,153.505
C06124=1093.423,402.371,-97.866,178.438,23.650,153.507
C06125=1093.430,402.618,-97.905,178.441,23.658,153.508
C06126=1093.435,402.864,-97.944,178.443,23.666,153.510
C06127=1093.441,403.111,-97.984,178.447,23.673,153.511
C06128=1093.447,403.359,-98.023,178.449,23.681,153.513
C06129=1093.454,403.605,-98.063,178.452,23.689,153.514
C06130=1093.460,403.851,-98.102,178.455,23.697,153.516
C06131=1093.466,404.098,-98.141,178.458,23.704,153.517
C06132=1093.472,404.345,-98.180,178.461,23.712,153.519
C06133=1093.478,404.593,-98.220,178.463,23.720,153.520
C06134=1093.484,404.839,-98.259,178.467,23.728,153.522
C06135=1093.490,405.086,-98.299,178.469,23.736,153.523
C06136=1093.496,405.333,-98.339,178.472,23.744,153.525
C06137=1093.502,405.580,-98.378,178.475,23.751,153.526
C06138=1093.508,405.826,-98.417,178.478,23.760,153.528
C06139=1093.514,406.073,-98.457,178.481,23.767,153.530
C06140=1093.520,406.320,-98.497,178.484,23.775,153.531
C06141=1093.526,406.567,-98.536,178.487,23.784,153.533
C06142=1093.533,406.814,-98.576,178.490,23.792,153.534
C06143=1093.538,407.060,-98.615,178.493,23.800,153.536
C06144=1093.544,407.306,-98.655,178.495,23.808,153.537
C06145=1093.551,407.554,-98.695,178.499,23.816,153.539
C06146=1093.557,407.801,-98.734,178.501,23.824,153.541
C06147=1093.563,408.047,-98.774,178.504,23.833,153.542
C06148=1093.569,408.294,-98.814,178.507,23.841,153.544
C06149=1093.575,408.540,-98.854,178.510,23.849,153.546
C06150=1093.581,408.787,-98.894,178.513,23.857,153.547
C06151=1093.587,409.034,-98.934,178.516,23.866,153.549
C06152=1093.593,409.281,-98.974,178.519,23.874,153.551
C06153=1093.599,409.528,-99.013,178.522,23.883,153.552
C06154=1093.605,409.774,-99.054,178.525,23.891,153.554
C06155=1093.612,410.021,-99.094,178.527,23.899,153.556
C06156=1093.616,410.268,-99.133,178.530,23.908,153.557
C06157=1093.623,410.489,-99.170,178.533,23.915,153.559
C06158=1093.628,410.711,-99.205,178.535,23.923,153.560
C06159=1093.633,410.933,-99.241,178.538,23.931,153.562
C06160=1093.639,411.154,-99.278,178.540,23.938,153.563
C06161=1093.644,411.375,-99.313,178.543,23.946,153.565
C06162=1093.650,411.597,-99.350,178.546,23.954,153.567
C06163=1093.655,411.819,-99.386,178.549,23.962,153.568
C06164=1093.660,412.041,-99.422,178.551,23.969,153.570
C06165=1093.667,412.287,-99.462,178.554,23.978,153.571
C06166=1093.673,412.534,-99.502,178.557,23.987,153.573
C06167=1093.679,412.780,-99.542,178.560,23.995,153.575
C06168=1093.685,413.027,-99.583,178.563,24.004,153.577
C06169=1093.691,413.274,-99.623,178.566,24.013,153.578
C06170=1093.698,413.520,-99.663,178.568,24.022,153.580
C06171=1093.703,413.767,-99.704,178.571,24.030,153.582
C06172=1093.710,414.014,-99.744,178.574,24.039,153.584
C06173=1093.716,414.260,-99.784,178.578,24.048,153.585
C06174=1093.722,414.507,-99.825,178.581,24.057,153.587
C06175=1093.729,414.754,-99.865,178.583,24.066,153.589
C06176=1093.735,415.001,-99.906,178.586,24.075,153.591
C06177=1093.741,415.247,-99.946,178.589,24.084,153.593
C06178=1093.748,415.493,-99.987,178.592,24.093,153.594
C06179=1093.754,415.740,-100.027,178.595,24.102,153.596
C06180=1093.760,415.987,-100.068,178.598,24.111,153.598
C06181=1093.766,416.233,-100.108,178.600,24.120,153.600
C06182=1093.772,416.480,-100.149,178.603,24.129,153.602
C06183=1093.778,416.726,-100.190,178.607,24.138,153.604
C06184=1093.784,416.973,-100.231,178.609,24.147,153.606
C06185=1093.791,417.220,-100.271,178.612,24.157,153.608
C06186=1093.797,417.466,-100.313,178.615,24.166,153.609
C06187=1093.802,417.713,-100.353,178.618,24.175,153.611
C06188=1093.809,417.960,-100.393,178.621,24.185,153.613
C06189=1093.815,418.206,-100.435,178.624,24.194,153.615
C06190=1093.821,418.452,-100.475,178.627,24.204,153.617
C06191=1093.827,418.698,-100.516,178.630,24.213,153.619
C06192=1093.833,418.946,-100.558,178.632,24.222,153.621
C06193=1093.840,419.192,-100.598,178.635,24.232,153.623
C06194=1093.846,419.439,-100.639,178.638,24.241,153.625
C06195=1093.852,419.685,-100.681,178.641,24.251,153.627
C06196=1093.858,419.931,-100.721,178.644,24.261,153.629
C06197=1093.865,420.178,-100.763,178.647,24.270,153.631
C06198=1093.870,420.425,-100.803,178.650,24.280,153.633
C06199=1093.877,420.671,-100.844,178.653,24.289,153.635
C06200=1093.883,420.917,-100.886,178.656,24.299,153.637
C06201=1093.889,421.165,-100.927,178.659,24.308,153.639
C06202=1093.895,421.411,-100.968,178.662,24.318,153.641
C06203=1093.902,421.657,-101.009,178.666,24.328,153.643
C06204=1093.908,421.904,-101.051,178.668,24.339,153.645
C06205=1093.914,422.151,-101.092,178.671,24.348,153.647
C06206=1093.921,422.396,-101.133,178.674,24.358,153.649
C06207=1093.927,422.643,-101.174,178.677,24.368,153.651
C06208=1093.933,422.890,-101.216,178.680,24.378,153.653
C06209=1093.939,423.136,-101.257,178.683,24.388,153.656
C06210=1093.945,423.382,-101.299,178.685,24.398,153.658
C06211=1093.952,423.629,-101.341,178.688,24.408,153.660
C06212=1093.957,423.875,-101.382,178.691,24.418,153.662
C06213=1093.963,424.104,-101.420,178.694,24.427,153.664
C06214=1093.969,424.333,-101.459,178.697,24.437,153.666
C06215=1093.974,424.562,-101.497,178.699,24.446,153.668
C06216=1093.980,424.791,-101.536,178.702,24.456,153.670
C06217=1093.986,425.020,-101.574,178.705,24.465,153.672
C06218=1093.992,425.249,-101.613,178.708,24.475,153.674
C06219=1093.998,425.478,-101.652,178.710,24.484,153.676
C06220=1094.003,425.706,-101.691,178.713,24.494,153.678
C06221=1094.010,425.953,-101.733,178.716,24.504,153.680
C06222=1094.016,426.199,-101.774,178.719,24.515,153.682
C06223=1094.022,426.445,-101.816,178.722,24.526,153.685
C06224=1094.029,426.692,-101.858,178.725,24.536,153.687
C06225=1094.035,426.938,-101.900,178.728,24.546,153.689
C06226=1094.041,427.185,-101.941,178.730,24.557,153.691
C06227=1094.047,427.431,-101.984,178.734,24.568,153.694
C06228=1094.054,427.677,-102.025,178.737,24.578,153.696
C06229=1094.060,427.924,-102.067,178.740,24.589,153.698
C06230=1094.067,428.170,-102.109,178.742,24.599,153.700
C06231=1094.073,428.416,-102.151,178.746,24.610,153.703
C06232=1094.080,428.662,-102.193,178.748,24.621,153.705
C06233=1094.085,428.909,-102.235,178.751,24.632,153.707
C06234=1094.092,429.155,-102.277,178.755,24.643,153.710
C06235=1094.098,429.401,-102.319,178.757,24.654,153.712
C06236=1094.104,429.648,-102.362,178.760,24.664,153.714
C06237=1094.110,429.894,-102.403,178.763,24.675,153.717
C06238=1094.117,430.140,-102.446,178.766,24.687,153.719
C06239=1094.123,430.386,-102.489,178.769,24.697,153.722
C06240=1094.129,430.633,-102.531,178.771,24.708,153.724
C06241=1094.136,430.879,-102.573,178.775,24.720,153.726
C06242=1094.142,431.125,-102.615,178.778,24.731,153.729
C06243=1094.148,431.371,-102.657,178.781,24.742,153.731
C06244=1094.154,431.618,-102.700,178.784,24.753,153.734
C06245=1094.161,431.864,-102.742,178.786,24.765,153.736
C06246=1094.167,432.110,-102.785,178.790,24.776,153.739
C06247=1094.173,432.357,-102.827,178.792,24.787,153.741
C06248=1094.180,432.603,-102.870,178.796,24.799,153.744
C06249=1094.186,432.849,-102.912,178.798,24.810,153.746
C06250=1094.193,433.095,-102.955,178.801,24.821,153.749
C06251=1094.199,433.341,-102.997,178.804,24.833,153.751
C06252=1094.205,433.587,-103.040,178.807,24.845,153.754
C06253=1094.212,433.834,-103.083,178.810,24.856,153.756
C06254=1094.217,434.080,-103.125,178.813,24.868,153.759
C06255=1094.224,434.326,-103.168,178.816,24.880,153.761
C06256=1094.230,434.572,-103.211,178.818,24.892,153.764
C06257=1094.236,434.818,-103.254,178.822,24.903,153.766
C06258=1094.243,435.065,-103.296,178.824,24.915,153.769
C06259=1094.249,435.311,-103.340,178.828,24.927,153.772
C06260=1094.255,435.556,-103.382,178.830,24.939,153.774
C06261=1094.261,435.803,-103.426,178.833,24.951,153.777
C06262=1094.268,436.049,-103.468,178.836,24.963,153.780
C06263=1094.274,436.295,-103.511,178.839,24.975,153.782
C06264=1094.280,436.541,-103.555,178.842,24.987,153.785
C06265=1094.287,436.787,-103.597,178.845,24.999,153.788
C06266=1094.293,437.034,-103.640,178.848,25.011,153.790
C06267=1094.300,437.279,-103.683,178.851,25.024,153.793
C06268=1094.306,437.525,-103.726,178.854,25.036,153.796
C06269=1094.312,437.755,-103.767,178.857,25.047,153.798
C06270=1094.318,437.985,-103.807,178.859,25.059,153.801
C06271=1094.324,438.216,-103.848,178.862,25.070,153.803
C06272=1094.330,438.446,-103.889,178.865,25.082,153.806
C06273=1094.336,438.676,-103.928,178.868,25.094,153.808
C06274=1094.342,438.905,-103.969,178.870,25.105,153.811
C06275=1094.348,439.136,-104.010,178.873,25.117,153.814
C06276=1094.354,439.366,-104.050,178.875,25.128,153.816
C06277=1094.361,439.612,-104.094,178.879,25.141,153.819
C06278=1094.368,439.858,-104.137,178.882,25.154,153.822
C06279=1094.374,440.105,-104.180,178.884,25.166,153.825
C06280=1094.380,440.351,-104.224,178.887,25.179,153.828
C06281=1094.386,440.596,-104.267,178.891,25.192,153.830
C06282=1094.393,440.842,-104.311,178.894,25.205,153.833
C06283=1094.400,441.088,-104.354,178.896,25.218,153.836
C06284=1094.406,441.334,-104.398,178.899,25.231,153.839
C06285=1094.412,441.580,-104.442,178.902,25.244,153.842
C06286=1094.419,441.826,-104.485,178.905,25.257,153.845
C06287=1094.425,442.072,-104.529,178.908,25.270,153.848
C06288=1094.432,442.318,-104.573,178.911,25.283,153.851
C06289=1094.438,442.564,-104.617,178.914,25.296,153.854
C06290=1094.444,442.810,-104.661,178.917,25.310,153.857
C06291=1094.451,443.056,-104.705,178.919,25.322,153.860
C06292=1094.457,443.302,-104.749,178.922,25.336,153.863
C06293=1094.464,443.548,-104.792,178.926,25.349,153.866
C06294=1094.470,443.794,-104.836,178.929,25.363,153.869
C06295=1094.477,444.040,-104.880,178.932,25.376,153.872
C06296=1094.483,444.286,-104.924,178.934,25.390,153.875
C06297=1094.490,444.531,-104.968,178.937,25.403,153.878
C06298=1094.496,444.777,-105.012,178.939,25.417,153.882
C06299=1094.503,445.023,-105.056,178.941,25.430,153.885
C06300=1094.509,445.269,-105.100,178.943,25.444,153.888
C06301=1094.516,445.514,-105.145,178.945,25.457,153.891
C06302=1094.522,445.760,-105.188,178.947,25.471,153.894
C06303=1094.529,446.007,-105.233,178.949,25.484,153.897
C06304=1094.535,446.253,-105.278,178.950,25.497,153.901
C06305=1094.542,446.499,-105.322,178.951,25.511,153.904
C06306=1094.548,446.745,-105.366,178.952,25.524,153.907
C06307=1094.555,446.990,-105.410,178.953,25.538,153.910
C06308=1094.561,447.236,-105.454,178.954,25.551,153.914
C06309=1094.567,447.482,-105.499,178.954,25.564,153.917
C06310=1094.574,447.728,-105.543,178.955,25.577,153.920
C06311=1094.581,447.974,-105.588,178.955,25.591,153.924
C06312=1094.587,448.220,-105.632,178.956,25.604,153.927
C06313=1094.593,448.465,-105.677,178.955,25.617,153.930
C06314=1094.600,448.712,-105.721,178.955,25.630,153.934
C06315=1094.607,448.957,-105.766,178.955,25.644,153.937
C06316=1094.614,449.203,-105.810,178.955,25.657,153.941
C06317=1094.620,449.449,-105.855,178.955,25.670,153.944
C06318=1094.626,449.694,-105.899,178.954,25.684,153.947
C06319=1094.633,449.940,-105.944,178.953,25.697,153.951
C06320=1094.641,450.187,-105.988,178.953,25.709,153.954
C06321=1094.252,450.178,-106.158,178.900,25.917,154.013
C06322=1094.244,449.932,-106.115,178.900,25.905,154.010
C06323=1094.238,449.686,-106.070,178.901,25.891,154.006
C06324=1094.231,449.441,-106.025,178.902,25.878,154.003
C06325=1094.224,449.195,-105.981,178.902,25.865,153.999
C06326=1094.217,448.949,-105.936,178.902,25.852,153.996
C06327=1094.211,448.703,-105.892,178.902,25.838,153.993
C06328=1094.205,448.458,-105.847,178.903,25.825,153.989
C06329=1094.198,448.211,-105.803,178.902,25.812,153.986
C06330=1094.191,447.966,-105.758,178.902,25.798,153.982
C06331=1094.185,447.720,-105.713,178.902,25.785,153.979
C06332=1094.179,447.474,-105.669,178.900,25.772,153.976
C06333=1094.171,447.228,-105.624,178.900,25.758,153.972
C06334=1094.165,446.982,-105.580,178.899,25.745,153.969
C06335=1094.159,446.736,-105.535,178.899,25.732,153.966
C06336=1094.152,446.490,-105.491,178.898,25.718,153.963
C06337=1094.146,446.245,-105.447,178.896,25.704,153.959
C06338=1094.139,445.998,-105.403,178.894,25.691,153.956
C06339=1094.133,445.753,-105.357,178.893,25.677,153.953
C06340=1094.126,445.507,-105.314,178.891,25.664,153.950
C06341=1094.120,445.261,-105.270,178.889,25.651,153.946
C06342=1094.113,445.015,-105.225,178.887,25.637,153.943
C06343=1094.107,444.769,-105.181,178.884,25.623,153.940
C06344=1094.100,444.523,-105.137,178.882,25.610,153.937
C06345=1094.093,444.278,-105.093,178.880,25.597,153.934
C06346=1094.086,444.031,-105.049,178.877,25.583,153.931
C06347=1094.080,443.785,-105.005,178.873,25.569,153.928
C06348=1094.074,443.539,-104.961,178.870,25.556,153.925
C06349=1094.067,443.293,-104.917,178.868,25.543,153.922
C06350=1094.061,443.047,-104.873,178.865,25.529,153.919
C06351=1094.054,442.802,-104.829,178.861,25.516,153.916
C06352=1094.048,442.556,-104.785,178.858,25.502,153.913
C06353=1094.041,442.310,-104.741,178.855,25.489,153.910
C06354=1094.035,442.064,-104.697,178.853,25.476,153.907
C06355=1094.028,441.818,-104.653,178.850,25.462,153.904
C06356=1094.022,441.572,-104.609,178.846,25.449,153.901
C06357=1094.015,441.326,-104.566,178.843,25.436,153.898
C06358=1094.009,441.080,-104.523,178.841,25.424,153.895
C06359=1094.003,440.834,-104.479,178.837,25.411,153.892
C06360=1093.996,440.588,-104.435,178.834,25.397,153.889
C06361=1093.990,440.343,-104.392,178.831,25.384,153.886
C06362=1093.984,440.097,-104.348,178.829,25.372,153.883
C06363=1093.977,439.851,-104.304,178.825,25.359,153.880
C06364=1093.971,439.604,-104.261,178.822,25.346,153.878
C06365=1093.964,439.358,-104.218,178.819,25.334,153.875
C06366=1093.958,439.134,-104.178,178.817,25.322,153.872
C06367=1093.952,438.908,-104.138,178.814,25.311,153.870
C06368=1093.946,438.683,-104.099,178.811,25.300,153.867
C06369=1093.940,438.458,-104.059,178.808,25.288,153.865
C06370=1093.934,438.234,-104.020,178.805,25.276,153.862
C06371=1093.928,438.009,-103.980,178.802,25.265,153.860
C06372=1093.922,437.785,-103.940,178.800,25.254,153.857
C06373=1093.916,437.560,-103.901,178.797,25.242,153.854
C06374=1093.910,437.314,-103.858,178.794,25.231,153.852
C06375=1093.904,437.068,-103.815,178.791,25.218,153.849
C06376=1093.897,436.822,-103.772,178.789,25.206,153.846
C06377=1093.891,436.575,-103.729,178.785,25.194,153.844
C06378=1093.885,436.329,-103.685,178.783,25.181,153.841
C06379=1093.878,436.084,-103.643,178.779,25.169,153.838
C06380=1093.872,435.837,-103.599,178.776,25.157,153.836
C06381=1093.865,435.591,-103.556,178.773,25.146,153.833
C06382=1093.859,435.345,-103.513,178.770,25.133,153.830
C06383=1093.853,435.099,-103.471,178.767,25.122,153.828
C06384=1093.847,434.853,-103.428,178.764,25.109,153.825
C06385=1093.840,434.606,-103.385,178.761,25.098,153.823
C06386=1093.834,434.361,-103.342,178.758,25.086,153.820
C06387=1093.828,434.115,-103.299,178.755,25.074,153.817
C06388=1093.821,433.868,-103.256,178.752,25.062,153.815
C06389=1093.815,433.622,-103.213,178.749,25.051,153.812
C06390=1093.809,433.376,-103.171,178.747,25.039,153.810
C06391=1093.802,433.129,-103.128,178.743,25.027,153.807
C06392=1093.796,432.884,-103.085,178.741,25.016,153.805
C06393=1093.789,432.638,-103.043,178.737,25.004,153.802
C06394=1093.783,432.391,-103.000,178.735,24.993,153.800
C06395=1093.777,432.145,-102.958,178.731,24.981,153.797
C06396=1093.770,431.899,-102.916,178.728,24.970,153.795
C06397=1093.764,431.652,-102.873,178.726,24.959,153.792
C06398=1093.758,431.406,-102.830,178.722,24.947,153.790
C06399=1093.751,431.160,-102.788,178.719,24.936,153.787
C06400=1093.746,430.914,-102.745,178.717,24.925,153.785
C06401=1093.739,430.667,-102.703,178.713,24.914,153.782
C06402=1093.732,430.421,-102.661,178.711,24.903,153.780
C06403=1093.726,430.175,-102.619,178.708,24.892,153.778
C06404=1093.720,429.929,-102.575,178.704,24.881,153.775
C06405=1093.714,429.683,-102.534,178.702,24.870,153.773
C06406=1093.707,429.436,-102.491,178.699,24.859,153.770
C06407=1093.701,429.190,-102.450,178.695,24.847,153.768
C06408=1093.695,428.944,-102.407,178.693,24.837,153.766
C06409=1093.689,428.697,-102.365,178.690,24.826,153.763
C06410=1093.682,428.451,-102.323,178.686,24.815,153.761
C06411=1093.676,428.204,-102.281,178.683,24.804,153.759
C06412=1093.669,427.959,-102.239,178.681,24.793,153.757
C06413=1093.663,427.712,-102.197,178.678,24.783,153.754
C06414=1093.657,427.466,-102.155,178.674,24.772,153.752
C06415=1093.650,427.219,-102.113,178.671,24.761,153.750
C06416=1093.644,426.973,-102.072,178.669,24.751,153.747
C06417=1093.638,426.727,-102.029,178.666,24.740,153.745
C06418=1093.631,426.480,-101.988,178.663,24.730,153.743
C06419=1093.625,426.234,-101.946,178.659,24.719,153.741
C06420=1093.618,425.988,-101.904,178.657,24.708,153.738
C06421=1093.613,425.742,-101.862,178.654,24.698,153.736
C06422=1093.607,425.512,-101.823,178.651,24.689,153.734
C06423=1093.601,425.283,-101.784,178.649,24.679,153.732
C06424=1093.595,425.054,-101.745,178.646,24.669,153.730
C06425=1093.589,424.824,-101.706,178.643,24.660,153.728
C06426=1093.583,424.595,-101.668,178.640,24.650,153.726
C06427=1093.578,424.365,-101.629,178.637,24.641,153.724
C06428=1093.572,424.136,-101.590,178.634,24.631,153.722
C06429=1093.566,423.907,-101.551,178.631,24.622,153.720
C06430=1093.560,423.660,-101.510,178.628,24.611,153.718
C06431=1093.554,423.414,-101.468,178.626,24.601,153.716
C06432=1093.548,423.167,-101.427,178.623,24.591,153.714
C06433=1093.542,422.921,-101.385,178.620,24.581,153.711
C06434=1093.536,422.675,-101.344,178.617,24.571,153.709
C06435=1093.528,422.428,-101.302,178.614,24.561,153.707
C06436=1093.523,422.181,-101.262,178.611,24.551,153.705
C06437=1093.517,421.935,-101.220,178.608,24.542,153.703
C06438=1093.510,421.688,-101.178,178.604,24.531,153.701
C06439=1093.504,421.442,-101.138,178.601,24.521,153.699
C06440=1093.498,421.196,-101.096,178.598,24.512,153.697
C06441=1093.491,420.949,-101.055,178.595,24.502,153.695
C06442=1093.485,420.702,-101.014,178.592,24.492,153.693
C06443=1093.479,420.457,-100.973,178.590,24.482,153.691
C06444=1093.473,420.210,-100.931,178.587,24.473,153.689
C06445=1093.467,419.963,-100.890,178.584,24.463,153.687
C06446=1093.460,419.717,-100.849,178.581,24.454,153.685
C06447=1093.454,419.470,-100.809,178.578,24.444,153.683
C06448=1093.448,419.224,-100.767,178.575,24.434,153.681
C06449=1093.442,418.978,-100.726,178.572,24.425,153.679
C06450=1093.435,418.731,-100.685,178.569,24.415,153.677
C06451=1093.429,418.484,-100.644,178.566,24.406,153.675
C06452=1093.423,418.238,-100.603,178.563,24.396,153.673
C06453=1093.417,417.992,-100.562,178.560,24.387,153.671
C06454=1093.411,417.745,-100.522,178.557,24.378,153.669
C06455=1093.405,417.498,-100.481,178.554,24.368,153.667
C06456=1093.399,417.251,-100.439,178.551,24.359,153.665
C06457=1093.392,417.005,-100.399,178.548,24.349,153.663
C06458=1093.387,416.758,-100.358,178.545,24.340,153.662
C06459=1093.381,416.512,-100.317,178.542,24.331,153.660
C06460=1093.374,416.265,-100.277,178.540,24.322,153.658
C06461=1093.368,416.019,-100.237,178.537,24.313,153.656
C06462=1093.362,415.773,-100.195,178.534,24.304,153.654
C06463=1093.355,415.525,-100.155,178.531,24.294,153.652
C06464=1093.349,415.279,-100.114,178.527,24.286,153.650
C06465=1093.343,415.032,-100.074,178.524,24.276,153.648
C06466=1093.336,414.785,-100.034,178.521,24.267,153.647
C06467=1093.331,414.539,-99.993,178.519,24.259,153.645
C06468=1093.324,414.293,-99.952,178.516,24.250,153.643
C06469=1093.318,414.046,-99.912,178.513,24.241,153.641
C06470=1093.312,413.799,-99.871,178.509,24.232,153.639
C06471=1093.306,413.553,-99.831,178.507,24.223,153.638
C06472=1093.299,413.306,-99.791,178.504,24.214,153.636
C06473=1093.293,413.059,-99.750,178.501,24.205,153.634
C06474=1093.287,412.812,-99.710,178.498,24.196,153.632
C06475=1093.280,412.566,-99.669,178.495,24.188,153.631
C06476=1093.275,412.319,-99.629,178.492,24.179,153.629
C06477=1093.268,412.073,-99.589,178.489,24.170,153.627
C06478=1093.263,411.851,-99.553,178.487,24.162,153.625
C06479=1093.258,411.628,-99.517,178.484,24.155,153.624
C06480=1093.253,411.406,-99.481,178.481,24.147,153.622
C06481=1093.246,411.185,-99.444,178.478,24.139,153.621
C06482=1093.241,410.962,-99.408,178.476,24.131,153.619
C06483=1093.236,410.741,-99.372,178.473,24.124,153.618
C06484=1093.230,410.518,-99.336,178.470,24.116,153.616
C06485=1093.225,410.296,-99.300,178.468,24.108,153.615
C06486=1093.218,410.050,-99.260,178.465,24.100,153.613
C06487=1093.213,409.803,-99.220,178.462,24.092,153.611
C06488=1093.207,409.556,-99.180,178.459,24.083,153.610
C06489=1093.200,409.309,-99.140,178.456,24.074,153.608
C06490=1093.194,409.063,-99.100,178.453,24.066,153.606
C06491=1093.189,408.815,-99.060,178.450,24.058,153.605
C06492=1093.182,408.569,-99.020,178.448,24.050,153.603
C06493=1093.177,408.322,-98.981,178.445,24.041,153.601
C06494=1093.170,408.076,-98.940,178.441,24.033,153.600
C06495=1093.164,407.829,-98.900,178.439,24.025,153.598
C06496=1093.158,407.582,-98.861,178.436,24.016,153.596
C06497=1093.152,407.335,-98.821,178.433,24.008,153.595
C06498=1093.145,407.089,-98.781,178.430,24.000,153.593
C06499=1093.140,406.842,-98.742,178.427,23.992,153.592
C06500=1093.134,406.596,-98.702,178.424,23.984,153.590
C06501=1093.128,406.348,-98.662,178.421,23.975,153.588
C06502=1093.122,406.102,-98.622,178.418,23.967,153.587
C06503=1093.116,405.855,-98.582,178.415,23.959,153.585
C06504=1093.110,405.607,-98.543,178.413,23.951,153.584
C06505=1093.103,405.362,-98.504,178.409,23.943,153.582
C06506=1093.097,405.115,-98.464,178.407,23.935,153.580
C06507=1093.091,404.868,-98.425,178.403,23.927,153.579
C06508=1093.085,404.620,-98.386,178.401,23.920,153.577
C06509=1093.079,404.375,-98.346,178.398,23.911,153.576
C06510=1093.073,404.128,-98.306,178.395,23.904,153.574
C06511=1093.067,403.880,-98.267,178.392,23.895,153.573
C06512=1093.061,403.633,-98.227,178.389,23.888,153.571
C06513=1093.056,403.387,-98.188,178.386,23.880,153.570
C06514=1093.049,403.140,-98.150,178.383,23.872,153.568
C06515=1093.042,402.893,-98.109,178.380,23.864,153.567
C06516=1093.036,402.646,-98.070,178.377,23.857,153.565
C06517=1093.031,402.400,-98.031,178.375,23.849,153.564
C06518=1093.025,402.153,-97.991,178.371,23.841,153.562
C06519=1093.018,401.906,-97.953,178.369,23.834,153.561
C06520=1093.012,401.660,-97.914,178.365,23.826,153.559
C06521=1093.006,401.412,-97.874,178.363,23.818,153.558
C06522=1093.000,401.165,-97.835,178.359,23.811,153.556
C06523=1092.994,400.919,-97.796,178.357,23.803,153.555
C06524=1092.988,400.672,-97.757,178.354,23.796,153.554
C06525=1092.982,400.424,-97.718,178.351,23.788,153.552
C06526=1092.977,400.178,-97.679,178.348,23.781,153.551
C06527=1092.970,399.931,-97.640,178.346,23.773,153.549
C06528=1092.964,399.685,-97.601,178.342,23.766,153.548
C06529=1092.958,399.437,-97.562,178.340,23.758,153.546
C06530=1092.952,399.191,-97.523,178.337,23.751,153.545
C06531=1092.946,398.944,-97.485,178.333,23.744,153.544
C06532=1092.940,398.697,-97.446,178.331,23.736,153.542
C06533=1092.934,398.450,-97.407,178.328,23.729,153.541
C06534=1092.929,398.229,-97.371,178.325,23.722,153.540
C06535=1092.923,398.007,-97.337,178.323,23.716,153.538
C06536=1092.918,397.785,-97.302,178.320,23.709,153.537
C06537=1092.912,397.563,-97.267,178.317,23.702,153.536
C06538=1092.907,397.342,-97.233,178.315,23.696,153.535
C06539=1092.901,397.120,-97.198,178.312,23.690,153.533
C06540=1092.896,396.898,-97.163,178.309,23.683,153.532
C06541=1092.890,396.677,-97.128,178.306,23.677,153.531
C06542=1092.885,396.430,-97.090,178.304,23.669,153.530
C06543=1092.878,396.183,-97.051,178.301,23.662,153.528
C06544=1092.873,395.936,-97.013,178.298,23.655,153.527
C06545=1092.866,395.689,-96.974,178.295,23.648,153.526
C06546=1092.861,395.442,-96.935,178.292,23.641,153.524
C06547=1092.855,395.196,-96.897,178.289,23.634,153.523
C06548=1092.849,394.948,-96.858,178.287,23.627,153.522
C06549=1092.843,394.702,-96.820,178.283,23.619,153.520
C06550=1092.837,394.454,-96.781,178.280,23.613,153.519
C06551=1092.831,394.208,-96.742,178.278,23.606,153.518
C06552=1092.824,393.961,-96.704,178.275,23.599,153.516
C06553=1092.819,393.714,-96.666,178.271,23.592,153.515
C06554=1092.812,393.467,-96.627,178.269,23.585,153.514
C06555=1092.806,393.220,-96.589,178.266,23.578,153.513
C06556=1092.801,392.973,-96.551,178.263,23.571,153.511
C06557=1092.794,392.726,-96.512,178.259,23.564,153.510
C06558=1092.788,392.479,-96.474,178.257,23.557,153.509
C06559=1092.783,392.232,-96.436,178.254,23.551,153.508
C06560=1092.776,391.985,-96.397,178.251,23.544,153.506
C06561=1092.770,391.739,-96.360,178.248,23.537,153.505
C06562=1092.764,391.491,-96.321,178.245,23.530,153.504
C06563=1092.758,391.245,-96.284,178.242,23.523,153.503
C06564=1092.752,390.998,-96.246,178.239,23.517,153.502
C06565=1092.746,390.751,-96.206,178.236,23.510,153.500
C06566=1092.740,390.504,-96.169,178.234,23.504,153.499
C06567=1092.734,390.257,-96.131,178.230,23.496,153.498
C06568=1092.728,390.010,-96.093,178.227,23.490,153.497
C06569=1092.722,389.763,-96.055,178.224,23.483,153.496
C06570=1092.716,389.516,-96.017,178.221,23.477,153.494
C06571=1092.709,389.269,-95.979,178.219,23.470,153.493
C06572=1092.703,389.022,-95.941,178.216,23.464,153.492
C06573=1092.698,388.775,-95.904,178.213,23.457,153.491
C06574=1092.692,388.529,-95.866,178.209,23.450,153.490
C06575=1092.685,388.281,-95.828,178.206,23.444,153.489
C06576=1092.679,388.034,-95.790,178.204,23.437,153.487
C06577=1092.673,387.788,-95.752,178.201,23.431,153.486
C06578=1092.668,387.541,-95.714,178.198,23.425,153.485
C06579=1092.662,387.294,-95.676,178.195,23.418,153.484
C06580=1092.656,387.046,-95.638,178.192,23.412,153.483
C06581=1092.650,386.799,-95.601,178.188,23.405,153.482
C06582=1092.644,386.552,-95.563,178.186,23.398,153.480
C06583=1092.638,386.306,-95.526,178.183,23.392,153.479
C06584=1092.632,386.059,-95.488,178.180,23.386,153.478
C06585=1092.627,385.812,-95.450,178.177,23.379,153.477
C06586=1092.620,385.564,-95.413,178.174,23.373,153.476
C06587=1092.614,385.317,-95.375,178.171,23.367,153.475
C06588=1092.609,385.070,-95.337,178.168,23.360,153.474
C06589=1092.602,384.824,-95.300,178.165,23.354,153.473
C06590=1092.598,384.608,-95.268,178.162,23.348,153.472
C06591=1092.592,384.392,-95.234,178.160,23.343,153.471
C06592=1092.587,384.178,-95.202,178.157,23.337,153.470
C06593=1092.582,383.963,-95.169,178.155,23.332,153.469
C06594=1092.577,383.748,-95.137,178.152,23.327,153.468
C06595=1092.572,383.533,-95.104,178.149,23.321,153.467
C06596=1092.566,383.318,-95.072,178.147,23.316,153.466
C06597=1092.562,383.103,-95.039,178.144,23.310,153.465
C06598=1092.556,382.856,-95.001,178.141,23.304,153.464
C06599=1092.550,382.609,-94.964,178.138,23.298,153.463
C06600=1092.543,382.361,-94.927,178.135,23.292,153.462
C06601=1092.537,382.114,-94.890,178.132,23.285,153.461
C06602=1092.532,381.867,-94.853,178.129,23.280,153.460
C06603=1092.526,381.620,-94.815,178.126,23.274,153.459
C06604=1092.519,381.373,-94.778,178.123,23.267,153.458
C06605=1092.514,381.126,-94.741,178.120,23.261,153.457
C06606=1092.508,380.879,-94.704,178.117,23.255,153.456
C06607=1092.502,380.632,-94.667,178.114,23.250,153.455
C06608=1092.496,380.385,-94.629,178.111,23.243,153.454
C06609=1092.490,380.138,-94.592,178.108,23.237,153.453
C06610=1092.484,379.891,-94.556,178.105,23.231,153.452
C06611=1092.478,379.644,-94.518,178.102,23.225,153.451
C06612=1092.472,379.397,-94.481,178.099,23.220,153.450
C06613=1092.466,379.149,-94.445,178.096,23.214,153.449
C06614=1092.460,378.903,-94.407,178.093,23.208,153.448
C06615=1092.454,378.655,-94.370,178.090,23.202,153.447
C06616=1092.448,378.408,-94.333,178.087,23.196,153.446
C06617=1092.443,378.161,-94.296,178.084,23.190,153.445
C06618=1092.436,377.914,-94.260,178.082,23.185,153.444
C06619=1092.431,377.667,-94.223,178.079,23.179,153.443
C06620=1092.425,377.420,-94.185,178.076,23.173,153.442
C06621=1092.418,377.173,-94.149,178.073,23.167,153.441
C06622=1092.413,376.925,-94.112,178.070,23.161,153.440
C06623=1092.406,376.678,-94.075,178.067,23.155,153.439
C06624=1092.401,376.431,-94.038,178.064,23.150,153.438
C06625=1092.395,376.184,-94.001,178.061,23.144,153.437
C06626=1092.389,375.937,-93.965,178.058,23.138,153.436
C06627=1092.383,375.689,-93.928,178.055,23.132,153.435
C06628=1092.378,375.443,-93.892,178.052,23.126,153.434
C06629=1092.372,375.195,-93.854,178.048,23.120,153.433
C06630=1092.366,374.948,-93.818,178.045,23.115,153.432
C06631=1092.360,374.701,-93.781,178.042,23.109,153.431
C06632=1092.354,374.454,-93.745,178.040,23.104,153.430
C06633=1092.348,374.206,-93.708,178.037,23.098,153.429
C06634=1092.342,373.959,-93.672,178.034,23.093,153.428
C06635=1092.336,373.712,-93.635,178.031,23.087,153.427
C06636=1092.330,373.465,-93.598,178.028,23.081,153.427
C06637=1092.324,373.218,-93.562,178.024,23.076,153.426
C06638=1092.319,372.971,-93.525,178.021,23.070,153.425
C06639=1092.313,372.723,-93.489,178.018,23.064,153.424
C06640=1092.306,372.476,-93.453,178.016,23.059,153.423
C06641=1092.301,372.229,-93.416,178.013,23.054,153.422
C06642=1092.294,371.982,-93.380,178.010,23.048,153.421
C06643=1092.288,371.734,-93.344,178.007,23.043,153.421
C06644=1092.283,371.488,-93.308,178.003,23.037,153.420
C06645=1092.277,371.240,-93.271,178.000,23.031,153.419
C06646=1092.268,370.837,-93.212,177.995,23.023,153.417
C06647=1092.258,370.435,-93.153,177.990,23.014,153.416
C06648=1092.248,370.032,-93.094,177.986,23.005,153.414
C06649=1092.239,369.629,-93.036,177.981,22.997,153.413
C06650=1092.233,369.382,-92.999,177.978,22.991,153.412
C06651=1092.227,369.134,-92.963,177.975,22.986,153.411
C06652=1092.221,368.887,-92.926,177.972,22.980,153.411
C06653=1092.215,368.640,-92.891,177.968,22.975,153.410
C06654=1092.210,368.393,-92.854,177.966,22.970,153.409
C06655=1092.204,368.145,-92.818,177.963,22.965,153.408
C06656=1092.197,367.898,-92.782,177.960,22.959,153.407
C06657=1092.192,367.651,-92.747,177.957,22.954,153.406
C06658=1092.186,367.403,-92.711,177.953,22.948,153.406
C06659=1092.180,367.156,-92.674,177.951,22.944,153.405
C06660=1092.175,366.909,-92.638,177.948,22.938,153.404
C06661=1092.169,366.661,-92.603,177.945,22.933,153.403
C06662=1092.162,366.414,-92.566,177.941,22.927,153.402
C06663=1092.157,366.167,-92.531,177.939,22.923,153.402
C06664=1092.151,365.920,-92.495,177.936,22.917,153.401
C06665=1092.145,365.673,-92.459,177.933,22.912,153.400
C06666=1092.139,365.426,-92.423,177.929,22.906,153.399
C06667=1092.133,365.178,-92.388,177.926,22.901,153.398
C06668=1092.127,364.930,-92.352,177.924,22.896,153.398
C06669=1092.122,364.683,-92.316,177.921,22.891,153.397
C06670=1092.116,364.436,-92.281,177.917,22.886,153.396
C06671=1092.109,364.189,-92.244,177.914,22.881,153.395
C06672=1092.104,363.942,-92.209,177.912,22.876,153.395
C06673=1092.098,363.694,-92.173,177.908,22.871,153.394
C06674=1092.092,363.446,-92.137,177.905,22.866,153.393
C06675=1092.086,363.199,-92.102,177.902,22.861,153.392
C06676=1092.080,362.952,-92.066,177.899,22.856,153.391
C06677=1092.074,362.704,-92.031,177.896,22.851,153.391
C06678=1092.069,362.457,-91.995,177.893,22.845,153.390
C06679=1092.063,362.209,-91.960,177.891,22.841,153.389
C06680=1092.057,361.962,-91.924,177.887,22.836,153.388
C06681=1092.051,361.715,-91.888,177.884,22.831,153.388
C06682=1092.045,361.467,-91.853,177.881,22.826,153.387
C06683=1092.039,361.220,-91.818,177.878,22.821,153.386
C06684=1092.033,360.973,-91.782,177.875,22.816,153.386
C06685=1092.028,360.726,-91.747,177.872,22.811,153.385
C06686=1092.022,360.478,-91.711,177.869,22.806,153.384
C06687=1092.017,360.230,-91.676,177.866,22.801,153.383
C06688=1092.011,359.983,-91.641,177.863,22.796,153.383
C06689=1092.004,359.735,-91.606,177.859,22.791,153.382
C06690=1091.998,359.488,-91.570,177.857,22.787,153.381
C06691=1091.992,359.241,-91.535,177.854,22.782,153.381
C06692=1091.987,358.993,-91.500,177.850,22.777,153.380
C06693=1091.980,358.746,-91.465,177.848,22.772,153.379
C06694=1091.975,358.499,-91.429,177.844,22.767,153.378
C06695=1091.969,358.251,-91.394,177.841,22.762,153.378
C06696=1091.964,358.003,-91.359,177.839,22.758,153.377
C06697=1091.957,357.756,-91.324,177.835,22.753,153.376
C06698=1091.948,357.369,-91.269,177.831,22.745,153.375
C06699=1091.939,356.981,-91.214,177.825,22.737,153.374
C06700=1091.930,356.594,-91.159,177.821,22.730,153.373
C06701=1091.921,356.207,-91.104,177.816,22.723,153.372
C06702=1091.915,355.959,-91.069,177.813,22.718,153.371
C06703=1091.909,355.712,-91.035,177.811,22.713,153.371
C06704=1091.903,355.464,-90.999,177.807,22.709,153.370
C06705=1091.898,355.216,-90.964,177.804,22.704,153.369
C06706=1091.892,354.970,-90.929,177.801,22.700,153.369
C06707=1091.886,354.721,-90.894,177.798,22.695,153.368
C06708=1091.880,354.475,-90.859,177.795,22.689,153.367
C06709=1091.874,354.227,-90.825,177.792,22.685,153.367
C06710=1091.869,353.979,-90.790,177.788,22.681,153.366
C06711=1091.863,353.732,-90.755,177.786,22.676,153.365
C06712=1091.857,353.484,-90.720,177.783,22.671,153.365
C06713=1091.851,353.237,-90.685,177.779,22.666,153.364
C06714=1091.845,352.989,-90.650,177.777,22.662,153.364
C06715=1091.839,352.742,-90.616,177.773,22.658,153.363
C06716=1091.834,352.495,-90.581,177.771,22.653,153.362
C06717=1091.827,352.247,-90.547,177.767,22.648,153.362
C06718=1091.822,351.999,-90.512,177.764,22.644,153.361
C06719=1091.816,351.751,-90.477,177.761,22.640,153.360
C06720=1091.810,351.504,-90.442,177.758,22.634,153.360
C06721=1091.804,351.257,-90.408,177.755,22.630,153.359
C06722=1091.798,351.009,-90.374,177.752,22.626,153.359
C06723=1091.793,350.761,-90.339,177.749,22.621,153.358
C06724=1091.787,350.514,-90.305,177.746,22.617,153.357
C06725=1091.781,350.266,-90.269,177.743,22.612,153.357
C06726=1091.775,350.019,-90.235,177.740,22.608,153.356
C06727=1091.769,349.772,-90.201,177.737,22.603,153.356
C06728=1091.764,349.524,-90.166,177.734,22.599,153.355
C06729=1091.758,349.276,-90.132,177.731,22.594,153.354
C06730=1091.752,349.029,-90.098,177.728,22.590,153.354
C06731=1091.746,348.781,-90.063,177.725,22.585,153.353
C06732=1091.740,348.533,-90.029,177.721,22.581,153.353
C06733=1091.734,348.286,-89.995,177.719,22.577,153.352
C06734=1091.729,348.039,-89.960,177.715,22.572,153.351
C06735=1091.723,347.791,-89.926,177.713,22.568,153.351
C06736=1091.717,347.543,-89.892,177.709,22.563,153.350
C06737=1091.712,347.296,-89.857,177.706,22.559,153.350
C06738=1091.706,347.048,-89.823,177.703,22.554,153.349
C06739=1091.699,346.800,-89.789,177.700,22.550,153.348
C06740=1091.694,346.553,-89.755,177.697,22.546,153.348
C06741=1091.688,346.306,-89.720,177.694,22.542,153.347
C06742=1091.683,346.058,-89.686,177.691,22.537,153.347
C06743=1091.676,345.810,-89.652,177.688,22.533,153.346
C06744=1091.671,345.562,-89.618,177.685,22.529,153.346
C06745=1091.665,345.315,-89.583,177.682,22.524,153.345
C06746=1091.660,345.067,-89.549,177.679,22.520,153.345
C06747=1091.654,344.820,-89.515,177.676,22.516,153.344
C06748=1091.648,344.572,-89.482,177.673,22.511,153.343
C06749=1091.642,344.324,-89.448,177.670,22.507,153.343
C06750=1091.632,343.939,-89.395,177.665,22.501,153.342
C06751=1091.624,343.555,-89.342,177.660,22.494,153.341
C06752=1091.615,343.170,-89.289,177.655,22.488,153.340
C06753=1091.606,342.785,-89.237,177.651,22.481,153.340
C06754=1091.600,342.537,-89.202,177.647,22.477,153.339
C06755=1091.594,342.290,-89.168,177.644,22.473,153.339
C06756=1091.588,342.042,-89.135,177.641,22.468,153.338
C06757=1091.582,341.795,-89.101,177.638,22.464,153.337
C06758=1091.577,341.548,-89.067,177.635,22.460,153.337
C06759=1091.571,341.300,-89.034,177.632,22.456,153.336
C06760=1091.565,341.052,-88.999,177.629,22.451,153.336
C06761=1091.559,340.804,-88.966,177.626,22.447,153.335
C06762=1091.553,340.556,-88.932,177.622,22.443,153.335
C06763=1091.548,340.309,-88.898,177.620,22.439,153.334
C06764=1091.542,340.061,-88.864,177.617,22.435,153.334
C06765=1091.536,339.813,-88.831,177.614,22.431,153.333
C06766=1091.531,339.565,-88.798,177.611,22.427,153.333
C06767=1091.525,339.318,-88.764,177.607,22.423,153.332
C06768=1091.519,339.070,-88.730,177.605,22.418,153.332
C06769=1091.513,338.823,-88.696,177.601,22.414,153.331
C06770=1091.508,338.575,-88.663,177.598,22.411,153.331
C06771=1091.502,338.327,-88.630,177.596,22.406,153.330
C06772=1091.496,338.080,-88.596,177.592,22.402,153.330
C06773=1091.490,337.831,-88.562,177.589,22.398,153.329
C06774=1091.484,337.584,-88.529,177.586,22.394,153.329
C06775=1091.478,337.336,-88.495,177.583,22.391,153.329
C06776=1091.473,337.088,-88.462,177.580,22.386,153.328
C06777=1091.467,336.841,-88.428,177.577,22.382,153.328
C06778=1091.461,336.593,-88.396,177.574,22.378,153.327
C06779=1091.455,336.346,-88.362,177.571,22.374,153.327
C06780=1091.449,336.098,-88.328,177.568,22.371,153.326
C06781=1091.444,335.850,-88.295,177.564,22.366,153.326
C06782=1091.438,335.602,-88.262,177.562,22.362,153.325
C06783=1091.432,335.354,-88.229,177.559,22.358,153.325
C06784=1091.426,335.106,-88.196,177.555,22.354,153.324
C06785=1091.420,334.859,-88.161,177.553,22.351,153.324
C06786=1091.415,334.611,-88.128,177.550,22.347,153.323
C06787=1091.409,334.364,-88.095,177.546,22.343,153.323
C06788=1091.403,334.116,-88.062,177.543,22.339,153.322
C06789=1091.397,333.868,-88.029,177.540,22.335,153.322
C06790=1091.391,333.620,-87.996,177.537,22.331,153.322
C06791=1091.386,333.373,-87.963,177.534,22.327,153.321
C06792=1091.381,333.125,-87.930,177.531,22.323,153.321
C06793=1091.375,332.877,-87.896,177.528,22.319,153.320
C06794=1091.369,332.630,-87.864,177.525,22.316,153.320
C06795=1091.363,332.382,-87.830,177.522,22.311,153.319
C06796=1091.358,332.134,-87.797,177.519,22.308,153.319
C06797=1091.351,331.886,-87.764,177.516,22.304,153.318
C06798=1091.346,331.638,-87.731,177.513,22.300,153.318
C06799=1091.340,331.391,-87.698,177.510,22.296,153.317
C06800=1091.334,331.143,-87.665,177.507,22.293,153.317
C06801=1091.328,330.895,-87.633,177.503,22.288,153.317
C06802=1091.319,330.505,-87.581,177.498,22.282,153.316
C06803=1091.310,330.114,-87.529,177.494,22.277,153.315
C06804=1091.300,329.723,-87.477,177.489,22.271,153.315
C06805=1091.291,329.332,-87.426,177.484,22.265,153.314
C06806=1091.285,329.084,-87.393,177.481,22.261,153.314
C06807=1091.279,328.837,-87.360,177.478,22.257,153.313
C06808=1091.273,328.589,-87.327,177.475,22.254,153.313
C06809=1091.268,328.341,-87.294,177.472,22.250,153.313
C06810=1091.261,328.093,-87.262,177.468,22.246,153.312
C06811=1091.256,327.845,-87.228,177.466,22.243,153.312
C06812=1091.250,327.598,-87.197,177.463,22.239,153.311
C06813=1091.244,327.350,-87.164,177.459,22.235,153.311
C06814=1091.239,327.102,-87.131,177.456,22.231,153.311
C06815=1091.233,326.854,-87.099,177.453,22.228,153.310
C06816=1091.226,326.606,-87.066,177.451,22.224,153.310
C06817=1091.221,326.358,-87.033,177.447,22.220,153.309
C06818=1091.215,326.111,-87.001,177.444,22.217,153.309
C06819=1091.209,325.863,-86.968,177.441,22.213,153.309
C06820=1091.204,325.615,-86.935,177.438,22.209,153.308
C06821=1091.198,325.367,-86.903,177.435,22.206,153.308
C06822=1091.192,325.120,-86.871,177.432,22.202,153.307
C06823=1091.186,324.872,-86.838,177.429,22.199,153.307
C06824=1091.181,324.624,-86.806,177.426,22.195,153.307
C06825=1091.174,324.376,-86.773,177.423,22.191,153.306
C06826=1091.169,324.129,-86.741,177.420,22.188,153.306
C06827=1091.163,323.881,-86.708,177.417,22.184,153.306
C06828=1091.157,323.632,-86.676,177.413,22.180,153.305
C06829=1091.151,323.384,-86.644,177.411,22.177,153.305
C06830=1091.146,323.137,-86.612,177.408,22.173,153.304
C06831=1091.140,322.889,-86.579,177.405,22.170,153.304
C06832=1091.134,322.641,-86.547,177.401,22.166,153.304
C06833=1091.129,322.394,-86.515,177.398,22.163,153.303
C06834=1091.123,322.145,-86.482,177.396,22.159,153.303
C06835=1091.118,321.897,-86.450,177.393,22.156,153.303
C06836=1091.112,321.650,-86.417,177.389,22.151,153.302
C06837=1091.106,321.402,-86.385,177.386,22.148,153.302
C06838=1091.100,321.154,-86.353,177.383,22.144,153.301
C06839=1091.094,320.907,-86.321,177.381,22.141,153.301
C06840=1091.089,320.658,-86.288,177.377,22.137,153.301
C06841=1091.083,320.410,-86.256,177.374,22.134,153.300
C06842=1091.078,320.162,-86.225,177.371,22.130,153.300
C06843=1091.072,319.914,-86.193,177.368,22.127,153.300
C06844=1091.066,319.667,-86.160,177.366,22.123,153.299
C06845=1091.060,319.419,-86.128,177.362,22.119,153.299
C06846=1091.055,319.171,-86.096,177.359,22.116,153.299
C06847=1091.049,318.923,-86.064,177.356,22.112,153.298
C06848=1091.043,318.675,-86.032,177.353,22.109,153.298
C06849=1091.038,318.427,-86.000,177.349,22.105,153.298
C06850=1091.032,318.179,-85.968,177.347,22.102,153.297
C06851=1091.027,317.932,-85.937,177.344,22.098,153.297
C06852=1091.021,317.683,-85.905,177.341,22.095,153.296
C06853=1091.016,317.436,-85.872,177.338,22.091,153.296
C06854=1091.007,317.038,-85.821,177.333,22.086,153.296
C06855=1090.997,316.640,-85.770,177.328,22.080,153.295
C06856=1090.988,316.243,-85.718,177.323,22.074,153.294
C06857=1090.979,315.845,-85.667,177.319,22.069,153.294
C06858=1090.974,315.598,-85.636,177.316,22.065,153.293
C06859=1090.968,315.350,-85.604,177.312,22.062,153.293
C06860=1090.963,315.102,-85.572,177.309,22.058,153.293
C06861=1090.957,314.853,-85.541,177.306,22.055,153.293
C06862=1090.951,314.606,-85.509,177.303,22.052,153.292
C06863=1090.945,314.358,-85.478,177.300,22.049,153.292
C06864=1090.939,314.110,-85.446,177.298,22.045,153.292
C06865=1090.933,313.862,-85.414,177.294,22.041,153.291
C06866=1090.928,313.615,-85.382,177.291,22.038,153.291
C06867=1090.922,313.366,-85.352,177.288,22.035,153.291
C06868=1090.916,313.118,-85.320,177.285,22.032,153.290
C06869=1090.910,312.870,-85.288,177.282,22.029,153.290
C06870=1090.903,312.622,-85.256,177.279,22.025,153.290
C06871=1090.898,312.374,-85.225,177.275,22.022,153.290
C06872=1090.892,312.126,-85.193,177.272,22.018,153.289
C06873=1090.886,311.879,-85.162,177.269,22.015,153.289
C06874=1090.881,311.631,-85.131,177.267,22.012,153.289
C06875=1090.875,311.383,-85.099,177.264,22.009,153.288
C06876=1090.869,311.135,-85.068,177.261,22.006,153.288
C06877=1090.863,310.887,-85.036,177.258,22.002,153.288
C06878=1090.858,310.639,-85.005,177.254,21.999,153.288
C06879=1090.851,310.391,-84.974,177.251,21.995,153.287
C06880=1090.846,310.144,-84.942,177.248,21.992,153.287
C06881=1090.841,309.895,-84.911,177.245,21.989,153.287
C06882=1090.834,309.648,-84.880,177.242,21.986,153.286
C06883=1090.829,309.399,-84.849,177.239,21.983,153.286
C06884=1090.822,309.152,-84.818,177.236,21.979,153.286
C06885=1090.817,308.903,-84.787,177.233,21.976,153.286
C06886=1090.812,308.656,-84.755,177.229,21.973,153.285
C06887=1090.805,308.407,-84.724,177.227,21.969,153.285
C06888=1090.800,308.160,-84.693,177.224,21.966,153.285
C06889=1090.794,307.912,-84.662,177.221,21.963,153.284
C06890=1090.788,307.664,-84.630,177.218,21.959,153.284
C06891=1090.783,307.416,-84.599,177.215,21.957,153.284
C06892=1090.777,307.168,-84.568,177.212,21.953,153.284
C06893=1090.771,306.920,-84.537,177.208,21.950,153.283
C06894=1090.765,306.672,-84.506,177.205,21.946,153.283
C06895=1090.760,306.424,-84.475,177.202,21.943,153.283
C06896=1090.754,306.176,-84.444,177.199,21.940,153.283
C06897=1090.748,305.928,-84.412,177.196,21.937,153.282
C06898=1090.743,305.680,-84.382,177.193,21.934,153.282
C06899=1090.737,305.432,-84.351,177.190,21.931,153.282
C06900=1090.731,305.184,-84.320,177.188,21.927,153.281
C06901=1090.726,304.936,-84.289,177.185,21.924,153.281
C06902=1090.720,304.688,-84.258,177.181,21.921,153.281
C06903=1090.714,304.441,-84.227,177.178,21.917,153.281
C06904=1090.708,304.192,-84.196,177.175,21.914,153.280
C06905=1090.703,303.944,-84.165,177.172,21.911,153.280
C06906=1090.694,303.550,-84.116,177.168,21.906,153.280
C06907=1090.685,303.154,-84.067,177.162,21.901,153.279
C06908=1090.676,302.760,-84.018,177.158,21.896,153.279
C06909=1090.667,302.364,-83.969,177.153,21.891,153.279
C06910=1090.661,302.117,-83.938,177.150,21.888,153.278
C06911=1090.656,301.869,-83.907,177.147,21.884,153.278
C06912=1090.650,301.621,-83.877,177.144,21.882,153.278
C06913=1090.645,301.373,-83.846,177.141,21.878,153.277
C06914=1090.639,301.125,-83.815,177.138,21.875,153.277
C06915=1090.633,300.876,-83.784,177.135,21.872,153.277
C06916=1090.628,300.629,-83.754,177.132,21.869,153.277
C06917=1090.622,300.381,-83.723,177.128,21.865,153.276
C06918=1090.617,300.133,-83.692,177.125,21.862,153.276
C06919=1090.611,299.885,-83.662,177.122,21.859,153.276
C06920=1090.606,299.637,-83.631,177.119,21.856,153.276
C06921=1090.600,299.389,-83.601,177.116,21.853,153.275
C06922=1090.594,299.141,-83.570,177.113,21.849,153.275
C06923=1090.589,298.893,-83.539,177.110,21.847,153.275
C06924=1090.583,298.645,-83.509,177.107,21.843,153.275
C06925=1090.577,298.397,-83.479,177.104,21.840,153.274
C06926=1090.572,298.149,-83.448,177.101,21.837,153.274
C06927=1090.566,297.900,-83.418,177.099,21.834,153.274
C06928=1090.560,297.652,-83.387,177.095,21.831,153.274
C06929=1090.555,297.404,-83.357,177.093,21.828,153.273
C06930=1090.550,297.156,-83.326,177.089,21.825,153.273
C06931=1090.544,296.908,-83.296,177.086,21.822,153.273
C06932=1090.538,296.661,-83.265,177.084,21.819,153.273
C06933=1090.532,296.412,-83.236,177.080,21.816,153.272
C06934=1090.527,296.164,-83.205,177.078,21.812,153.272
C06935=1090.521,295.916,-83.175,177.074,21.810,153.272
C06936=1090.515,295.669,-83.145,177.071,21.807,153.272
C06937=1090.509,295.420,-83.115,177.068,21.803,153.272
C06938=1090.504,295.172,-83.085,177.065,21.801,153.271
C06939=1090.498,294.924,-83.053,177.062,21.798,153.271
C06940=1090.492,294.676,-83.023,177.059,21.794,153.271
C06941=1090.487,294.427,-82.993,177.056,21.792,153.271
C06942=1090.481,294.179,-82.963,177.053,21.789,153.271
C06943=1090.475,293.932,-82.933,177.050,21.785,153.270
C06944=1090.469,293.683,-82.903,177.047,21.783,153.270
C06945=1090.464,293.435,-82.873,177.044,21.780,153.270
C06946=1090.458,293.187,-82.843,177.041,21.776,153.270
C06947=1090.452,292.939,-82.813,177.038,21.774,153.269
C06948=1090.446,292.691,-82.782,177.035,21.771,153.269
C06949=1090.441,292.443,-82.753,177.032,21.767,153.269
C06950=1090.435,292.195,-82.722,177.029,21.765,153.269
C06951=1090.430,291.947,-82.693,177.026,21.762,153.269
C06952=1090.424,291.699,-82.662,177.023,21.758,153.268
C06953=1090.418,291.450,-82.633,177.020,21.756,153.268
C06954=1090.413,291.203,-82.602,177.017,21.753,153.268
C06955=1090.407,290.954,-82.573,177.014,21.750,153.268
C06956=1090.401,290.706,-82.542,177.011,21.747,153.267
C06957=1090.395,290.458,-82.513,177.008,21.744,153.267
C06958=1090.387,290.077,-82.467,177.004,21.739,153.267
C06959=1090.378,289.696,-82.421,176.998,21.734,153.267
C06960=1090.370,289.315,-82.376,176.994,21.730,153.266
C06961=1090.361,288.935,-82.330,176.989,21.726,153.266
C06962=1090.355,288.687,-82.301,176.986,21.722,153.266
C06963=1090.349,288.438,-82.271,176.983,21.720,153.266
C06964=1090.343,288.190,-82.241,176.980,21.717,153.266
C06965=1090.338,287.942,-82.211,176.977,21.714,153.265
C06966=1090.331,287.694,-82.182,176.975,21.711,153.265
C06967=1090.326,287.446,-82.152,176.972,21.709,153.265
C06968=1090.320,287.198,-82.122,176.969,21.706,153.265
C06969=1090.315,286.950,-82.093,176.966,21.702,153.265
C06970=1090.309,286.702,-82.064,176.963,21.700,153.264
C06971=1090.303,286.453,-82.034,176.960,21.697,153.264
C06972=1090.298,286.205,-82.004,176.956,21.694,153.264
C06973=1090.292,285.957,-81.974,176.953,21.691,153.264
C06974=1090.286,285.709,-81.945,176.950,21.688,153.264
C06975=1090.280,285.460,-81.915,176.947,21.685,153.264
C06976=1090.275,285.212,-81.886,176.944,21.682,153.263
C06977=1090.269,284.965,-81.857,176.941,21.679,153.263
C06978=1090.263,284.717,-81.827,176.938,21.676,153.263
C06979=1090.258,284.468,-81.797,176.935,21.673,153.263
C06980=1090.252,284.220,-81.768,176.932,21.671,153.263
C06981=1090.246,283.972,-81.739,176.929,21.668,153.262
C06982=1090.241,283.723,-81.709,176.926,21.665,153.262
C06983=1090.236,283.476,-81.680,176.924,21.662,153.262
C06984=1090.229,283.227,-81.651,176.921,21.660,153.262
C06985=1090.224,282.979,-81.621,176.918,21.657,153.262
C06986=1090.218,282.731,-81.591,176.915,21.654,153.262
C06987=1090.213,282.483,-81.563,176.912,21.651,153.261
C06988=1090.207,282.235,-81.533,176.909,21.648,153.261
C06989=1090.202,281.986,-81.503,176.906,21.645,153.261
C06990=1090.196,281.738,-81.474,176.902,21.642,153.261
C06991=1090.190,281.490,-81.445,176.899,21.639,153.261
C06992=1090.185,281.242,-81.417,176.896,21.636,153.260
C06993=1090.179,280.993,-81.387,176.893,21.633,153.260
C06994=1090.173,280.745,-81.358,176.890,21.631,153.260
C06995=1090.167,280.497,-81.328,176.888,21.628,153.260
C06996=1090.162,280.249,-81.300,176.885,21.625,153.260
C06997=1090.156,280.001,-81.270,176.882,21.622,153.260
C06998=1090.150,279.753,-81.241,176.879,21.620,153.259
C06999=1090.145,279.503,-81.212,176.876,21.617,153.259
C07000=1090.139,279.256,-81.183,176.873,21.614,153.259
C07001=1090.134,279.008,-81.154,176.870,21.611,153.259
C07002=1090.127,278.759,-81.125,176.867,21.608,153.259
C07003=1090.122,278.510,-81.096,176.863,21.605,153.259
C07004=1090.117,278.263,-81.067,176.860,21.602,153.258
C07005=1090.111,278.015,-81.038,176.858,21.600,153.258
C07006=1090.105,277.766,-81.009,176.855,21.597,153.258
C07007=1090.099,277.518,-80.981,176.852,21.594,153.258
C07008=1090.094,277.270,-80.951,176.849,21.592,153.258
C07009=1090.088,277.022,-80.922,176.846,21.589,153.258
C07010=1090.080,276.650,-80.879,176.841,21.585,153.257
C07011=1090.071,276.279,-80.835,176.837,21.581,153.257
C07012=1090.062,275.907,-80.793,176.833,21.577,153.257
C07013=1090.054,275.536,-80.750,176.828,21.572,153.257
C07014=1090.048,275.287,-80.721,176.825,21.570,153.257
C07015=1090.043,275.039,-80.692,176.822,21.567,153.256
C07016=1090.037,274.791,-80.663,176.819,21.564,153.256
C07017=1090.031,274.544,-80.634,176.816,21.561,153.256
C07018=1090.026,274.295,-80.605,176.814,21.559,153.256
C07019=1090.020,274.046,-80.576,176.810,21.556,153.256
C07020=1090.015,273.798,-80.548,176.807,21.553,153.256
C07021=1090.009,273.550,-80.520,176.804,21.551,153.256
C07022=1090.003,273.301,-80.490,176.801,21.548,153.255
C07023=1089.998,273.053,-80.462,176.798,21.545,153.255
C07024=1089.992,272.805,-80.433,176.795,21.542,153.255
C07025=1089.986,272.557,-80.405,176.793,21.540,153.255
C07026=1089.981,272.308,-80.376,176.790,21.537,153.255
C07027=1089.975,272.060,-80.347,176.787,21.534,153.255
C07028=1089.969,271.812,-80.320,176.784,21.531,153.255
C07029=1089.963,271.564,-80.290,176.781,21.529,153.254
C07030=1089.958,271.315,-80.263,176.777,21.526,153.254
C07031=1089.952,271.067,-80.234,176.775,21.524,153.254
C07032=1089.947,270.819,-80.205,176.772,21.521,153.254
C07033=1089.941,270.570,-80.177,176.769,21.518,153.254
C07034=1089.935,270.321,-80.148,176.766,21.515,153.254
C07035=1089.930,270.073,-80.120,176.763,21.512,153.253
C07036=1089.924,269.825,-80.091,176.760,21.510,153.253
C07037=1089.918,269.577,-80.063,176.757,21.508,153.253
C07038=1089.912,269.328,-80.035,176.754,21.505,153.253
C07039=1089.907,269.080,-80.007,176.751,21.502,153.253
C07040=1089.901,268.832,-79.977,176.748,21.499,153.253
C07041=1089.896,268.584,-79.949,176.745,21.497,153.253
C07042=1089.890,268.335,-79.921,176.742,21.494,153.253
C07043=1089.885,268.087,-79.893,176.740,21.491,153.252
C07044=1089.879,267.838,-79.865,176.737,21.488,153.252
C07045=1089.874,267.590,-79.837,176.733,21.486,153.252
C07046=1089.867,267.342,-79.808,176.730,21.483,153.252
C07047=1089.862,267.094,-79.780,176.727,21.480,153.252
C07048=1089.856,266.845,-79.752,176.725,21.478,153.252
C07049=1089.851,266.597,-79.724,176.722,21.476,153.252
C07050=1089.845,266.349,-79.695,176.719,21.473,153.252
C07051=1089.839,266.101,-79.667,176.716,21.470,153.251
C07052=1089.833,265.852,-79.639,176.713,21.467,153.251
C07053=1089.828,265.604,-79.611,176.710,21.465,153.251
C07054=1089.822,265.355,-79.583,176.707,21.462,153.251
C07055=1089.817,265.107,-79.555,176.704,21.459,153.251
C07056=1089.811,264.858,-79.526,176.701,21.456,153.251
C07057=1089.805,264.610,-79.498,176.698,21.454,153.251
C07058=1089.800,264.362,-79.471,176.696,21.452,153.251
C07059=1089.793,264.114,-79.443,176.693,21.449,153.250
C07060=1089.788,263.866,-79.415,176.689,21.446,153.250
C07061=1089.782,263.617,-79.387,176.686,21.443,153.250
C07062=1089.774,263.248,-79.345,176.682,21.440,153.250
C07063=1089.765,262.879,-79.305,176.678,21.436,153.250
C07064=1089.757,262.511,-79.263,176.673,21.432,153.250
C07065=1089.747,262.142,-79.222,176.669,21.429,153.250
C07066=1089.742,261.894,-79.194,176.666,21.426,153.249
C07067=1089.736,261.645,-79.166,176.663,21.423,153.249
C07068=1089.731,261.397,-79.138,176.660,21.421,153.249
C07069=1089.725,261.149,-79.111,176.657,21.418,153.249
C07070=1089.717,260.802,-79.072,176.653,21.414,153.249
C07071=1089.709,260.456,-79.033,176.649,21.411,153.249
C07072=1089.700,260.110,-78.994,176.645,21.408,153.249
C07073=1089.693,259.764,-78.956,176.641,21.404,153.249
C07074=1089.687,259.514,-78.928,176.638,21.401,153.248
C07075=1089.681,259.267,-78.901,176.635,21.398,153.248
C07076=1089.676,259.019,-78.873,176.632,21.396,153.248
C07077=1089.670,258.769,-78.845,176.629,21.394,153.248
C07078=1089.664,258.521,-78.818,176.626,21.391,153.248
C07079=1089.659,258.273,-78.790,176.623,21.388,153.248
C07080=1089.652,258.024,-78.763,176.620,21.386,153.248
C07081=1089.647,257.776,-78.735,176.618,21.384,153.248
C07082=1089.642,257.528,-78.707,176.615,21.381,153.248
C07083=1089.635,257.279,-78.680,176.611,21.378,153.248
C07084=1089.630,257.030,-78.652,176.608,21.375,153.247
C07085=1089.624,256.783,-78.625,176.606,21.374,153.247
C07086=1089.619,256.533,-78.597,176.603,21.371,153.247
C07087=1089.613,256.285,-78.570,176.600,21.368,153.247
C07088=1089.608,256.037,-78.543,176.596,21.365,153.247
C07089=1089.602,255.789,-78.515,176.594,21.363,153.247
C07090=1089.596,255.540,-78.488,176.591,21.361,153.247
C07091=1089.590,255.292,-78.460,176.588,21.358,153.247
C07092=1089.585,255.043,-78.433,176.585,21.355,153.246
C07093=1089.579,254.795,-78.405,176.583,21.353,153.246
C07094=1089.574,254.546,-78.378,176.579,21.350,153.246
C07095=1089.568,254.298,-78.350,176.576,21.348,153.246
C07096=1089.563,254.050,-78.323,176.574,21.345,153.246
C07097=1089.557,253.801,-78.296,176.571,21.342,153.246
C07098=1089.551,253.553,-78.268,176.568,21.340,153.246
C07099=1089.545,253.304,-78.242,176.565,21.337,153.246
C07100=1089.540,253.055,-78.214,176.562,21.335,153.246
C07101=1089.534,252.808,-78.187,176.559,21.332,153.246
C07102=1089.529,252.559,-78.160,176.556,21.329,153.245
C07103=1089.523,252.310,-78.133,176.553,21.327,153.245
C07104=1089.518,252.061,-78.105,176.551,21.325,153.245
C07105=1089.511,251.814,-78.078,176.548,21.322,153.245
C07106=1089.506,251.565,-78.051,176.544,21.319,153.245
C07107=1089.501,251.317,-78.024,176.542,21.317,153.245
C07108=1089.496,251.068,-77.997,176.539,21.315,153.245
C07109=1089.490,250.820,-77.970,176.536,21.312,153.245
C07110=1089.484,250.571,-77.942,176.534,21.309,153.244
C07111=1089.478,250.322,-77.915,176.531,21.307,153.244
C07112=1089.473,250.074,-77.888,176.528,21.304,153.244
C07113=1089.467,249.825,-77.861,176.524,21.302,153.244
C07114=1089.462,249.552,-77.831,176.521,21.299,153.244
C07115=1089.455,249.278,-77.802,176.518,21.296,153.244
C07116=1089.449,249.005,-77.772,176.515,21.293,153.244
C07117=1089.444,248.731,-77.742,176.512,21.290,153.244
C07118=1089.438,248.483,-77.715,176.509,21.288,153.244
C07119=1089.432,248.234,-77.689,176.507,21.285,153.244
C07120=1089.427,247.986,-77.661,176.504,21.282,153.243
C07121=1089.421,247.737,-77.635,176.500,21.280,153.243
C07122=1089.416,247.489,-77.607,176.498,21.278,153.243
C07123=1089.410,247.241,-77.580,176.495,21.275,153.243
C07124=1089.404,246.992,-77.553,176.492,21.272,153.243
C07125=1089.399,246.742,-77.527,176.489,21.270,153.243
C07126=1089.393,246.494,-77.500,176.486,21.267,153.243
C07127=1089.387,246.246,-77.473,176.483,21.265,153.243
C07128=1089.382,245.997,-77.447,176.481,21.263,153.243
C07129=1089.377,245.749,-77.419,176.478,21.260,153.243
C07130=1089.371,245.500,-77.393,176.475,21.257,153.242
C07131=1089.365,245.252,-77.366,176.473,21.255,153.242
C07132=1089.359,245.004,-77.340,176.469,21.253,153.242
C07133=1089.354,244.755,-77.312,176.466,21.250,153.242
C07134=1089.348,244.507,-77.286,176.464,21.248,153.242
C07135=1089.343,244.258,-77.259,176.461,21.245,153.242
C07136=1089.337,244.009,-77.233,176.458,21.242,153.242
C07137=1089.331,243.761,-77.206,176.455,21.240,153.242
C07138=1089.326,243.512,-77.179,176.452,21.238,153.242
C07139=1089.321,243.264,-77.153,176.449,21.235,153.242
C07140=1089.315,243.015,-77.126,176.447,21.233,153.241
C07141=1089.309,242.767,-77.100,176.444,21.230,153.241
C07142=1089.304,242.518,-77.073,176.440,21.228,153.241
C07143=1089.298,242.270,-77.047,176.438,21.225,153.241
C07144=1089.292,242.021,-77.020,176.435,21.223,153.241
C07145=1089.287,241.772,-76.994,176.432,21.220,153.241
C07146=1089.281,241.524,-76.967,176.430,21.218,153.241
C07147=1089.275,241.276,-76.941,176.426,21.216,153.241
C07148=1089.269,241.027,-76.914,176.423,21.213,153.241
C07149=1089.264,240.778,-76.888,176.421,21.211,153.241
C07150=1089.258,240.530,-76.862,176.418,21.208,153.241
C07151=1089.252,240.282,-76.835,176.415,21.206,153.241
C07152=1089.247,240.033,-76.809,176.412,21.203,153.240
C07153=1089.241,239.784,-76.782,176.409,21.201,153.240
C07154=1089.236,239.535,-76.756,176.407,21.199,153.240
C07155=1089.230,239.287,-76.730,176.404,21.196,153.240
C07156=1089.224,239.039,-76.703,176.401,21.193,153.240
C07157=1089.219,238.790,-76.677,176.398,21.191,153.240
C07158=1089.213,238.541,-76.650,176.395,21.189,153.240
C07159=1089.207,238.292,-76.625,176.392,21.186,153.240
C07160=1089.202,238.044,-76.598,176.390,21.184,153.240
C07161=1089.196,237.795,-76.572,176.386,21.181,153.240
C07162=1089.190,237.547,-76.545,176.384,21.179,153.240
C07163=1089.185,237.298,-76.519,176.381,21.177,153.240
C07164=1089.178,237.050,-76.493,176.378,21.174,153.239
C07165=1089.173,236.801,-76.468,176.376,21.172,153.239
C07166=1089.165,236.423,-76.428,176.371,21.168,153.239
C07167=1089.156,236.045,-76.388,176.367,21.164,153.239
C07168=1089.148,235.666,-76.348,176.362,21.160,153.239
C07169=1089.140,235.288,-76.308,176.358,21.157,153.239
C07170=1089.134,235.039,-76.282,176.355,21.154,153.239
C07171=1089.128,234.790,-76.257,176.353,21.152,153.239
C07172=1089.122,234.542,-76.230,176.350,21.150,153.239
C07173=1089.117,234.293,-76.204,176.347,21.147,153.239
C07174=1089.111,234.044,-76.178,176.344,21.145,153.239
C07175=1089.106,233.796,-76.152,176.341,21.142,153.238
C07176=1089.101,233.547,-76.126,176.339,21.140,153.238
C07177=1089.094,233.299,-76.101,176.336,21.137,153.238
C07178=1089.089,233.050,-76.074,176.333,21.135,153.238
C07179=1089.083,232.801,-76.048,176.330,21.132,153.238
C07180=1089.078,232.552,-76.022,176.327,21.130,153.238
C07181=1089.072,232.304,-75.997,176.325,21.128,153.238
C07182=1089.066,232.056,-75.971,176.322,21.125,153.238
C07183=1089.061,231.807,-75.945,176.319,21.123,153.238
C07184=1089.055,231.558,-75.919,176.316,21.120,153.238
C07185=1089.049,231.309,-75.893,176.313,21.118,153.238
C07186=1089.044,231.061,-75.868,176.311,21.115,153.237
C07187=1089.039,230.812,-75.842,176.308,21.113,153.237
C07188=1089.032,230.564,-75.816,176.305,21.111,153.237
C07189=1089.027,230.315,-75.790,176.302,21.108,153.237
C07190=1089.022,230.067,-75.764,176.299,21.106,153.237
C07191=1089.016,229.818,-75.739,176.297,21.104,153.237
C07192=1089.010,229.569,-75.713,176.294,21.101,153.237
C07193=1089.004,229.320,-75.688,176.291,21.099,153.237
C07194=1088.999,229.072,-75.662,176.288,21.096,153.237
C07195=1088.993,228.823,-75.637,176.286,21.094,153.237
C07196=1088.988,228.574,-75.611,176.283,21.092,153.237
C07197=1088.981,228.326,-75.585,176.280,21.089,153.237
C07198=1088.977,228.078,-75.560,176.277,21.087,153.237
C07199=1088.971,227.829,-75.534,176.274,21.084,153.237
C07200=1088.965,227.580,-75.509,176.272,21.082,153.236
C07201=1088.959,227.331,-75.483,176.269,21.080,153.236
C07202=1088.954,227.083,-75.458,176.266,21.078,153.236
C07203=1088.948,226.834,-75.432,176.263,21.075,153.236
C07204=1088.942,226.585,-75.406,176.261,21.073,153.236
C07205=1088.937,226.336,-75.381,176.258,21.070,153.236
C07206=1088.931,226.088,-75.356,176.255,21.068,153.236
C07207=1088.926,225.839,-75.330,176.252,21.066,153.236
C07208=1088.919,225.591,-75.304,176.250,21.063,153.236
C07209=1088.915,225.342,-75.279,176.247,21.061,153.236
C07210=1088.909,225.093,-75.254,176.243,21.058,153.236
C07211=1088.903,224.844,-75.228,176.241,21.056,153.236
C07212=1088.898,224.596,-75.203,176.238,21.054,153.236
C07213=1088.891,224.347,-75.178,176.236,21.051,153.236
C07214=1088.887,224.099,-75.152,176.233,21.049,153.235
C07215=1088.880,223.851,-75.127,176.230,21.047,153.235
C07216=1088.875,223.601,-75.102,176.227,21.044,153.235
C07217=1088.870,223.353,-75.077,176.225,21.042,153.235
C07218=1088.861,222.966,-75.038,176.220,21.038,153.235
C07219=1088.853,222.579,-74.998,176.216,21.034,153.235
C07220=1088.844,222.192,-74.958,176.212,21.030,153.235
C07221=1088.835,221.805,-74.919,176.208,21.027,153.235
C07222=1088.829,221.556,-74.894,176.205,21.025,153.235
C07223=1088.823,221.307,-74.869,176.202,21.022,153.235
C07224=1088.818,221.059,-74.844,176.199,21.020,153.235
C07225=1088.812,220.810,-74.818,176.197,21.018,153.235
C07226=1088.806,220.561,-74.794,176.194,21.015,153.234
C07227=1088.800,220.313,-74.769,176.191,21.013,153.234
C07228=1088.795,220.063,-74.744,176.188,21.011,153.234
C07229=1088.790,219.815,-74.719,176.186,21.008,153.234
C07230=1088.784,219.567,-74.693,176.183,21.006,153.234
C07231=1088.778,219.318,-74.669,176.180,21.004,153.234
C07232=1088.773,219.069,-74.643,176.177,21.001,153.234
C07233=1088.767,218.820,-74.618,176.175,20.999,153.234
C07234=1088.761,218.572,-74.593,176.172,20.997,153.234
C07235=1088.755,218.323,-74.569,176.170,20.994,153.234
C07236=1088.750,218.075,-74.544,176.166,20.992,153.234
C07237=1088.745,217.825,-74.519,176.164,20.990,153.234
C07238=1088.739,217.577,-74.494,176.161,20.987,153.234
C07239=1088.733,217.328,-74.469,176.159,20.985,153.234
C07240=1088.727,217.080,-74.444,176.155,20.983,153.234
C07241=1088.722,216.831,-74.420,176.153,20.980,153.233
C07242=1088.716,216.583,-74.395,176.150,20.978,153.233
C07243=1088.711,216.333,-74.369,176.148,20.976,153.233
C07244=1088.705,216.085,-74.344,176.145,20.973,153.233
C07245=1088.699,215.836,-74.320,176.142,20.971,153.233
C07246=1088.694,215.587,-74.295,176.139,20.968,153.233
C07247=1088.688,215.338,-74.270,176.137,20.966,153.233
C07248=1088.683,215.090,-74.246,176.134,20.964,153.233
C07249=1088.677,214.840,-74.221,176.131,20.961,153.233
C07250=1088.672,214.592,-74.196,176.129,20.959,153.233
C07251=1088.666,214.344,-74.171,176.126,20.957,153.233
C07252=1088.661,214.094,-74.147,176.124,20.954,153.233
C07253=1088.655,213.846,-74.122,176.120,20.952,153.233
C07254=1088.649,213.597,-74.097,176.118,20.950,153.232
C07255=1088.644,213.349,-74.073,176.115,20.947,153.232
C07256=1088.638,213.101,-74.048,176.113,20.945,153.232
C07257=1088.632,212.851,-74.023,176.110,20.942,153.232
C07258=1088.627,212.603,-73.999,176.107,20.940,153.232
C07259=1088.621,212.353,-73.974,176.104,20.938,153.232
C07260=1088.615,212.105,-73.950,176.102,20.936,153.232
C07261=1088.610,211.856,-73.925,176.099,20.933,153.232
C07262=1088.604,211.608,-73.901,176.096,20.931,153.232
C07263=1088.599,211.359,-73.876,176.094,20.929,153.232
C07264=1088.593,211.110,-73.852,176.091,20.926,153.232
C07265=1088.588,210.861,-73.827,176.088,20.924,153.232
C07266=1088.582,210.612,-73.802,176.085,20.921,153.232
C07267=1088.576,210.364,-73.778,176.083,20.920,153.232
C07268=1088.571,210.115,-73.754,176.080,20.917,153.232
C07269=1088.565,209.866,-73.729,176.078,20.915,153.232
C07270=1088.557,209.483,-73.692,176.074,20.911,153.231
C07271=1088.548,209.100,-73.654,176.069,20.907,153.231
